LIN {X 0,Y 216.185,Z 698.743,A -85,B 0,C 180,E1 -24874.885,E2 -24874.885} C_VEL
LIN {X 0,Y 219.913,Z 693.734,A -85,B 0,C 180,E1 -24875.576,E2 -24875.576} C_VEL
LIN {X 0,Y 220.4,Z 693.095,A -85,B 0,C 180,E1 -24876,E2 -24876} C_VEL
LIN {X 0,Y 211.801,Z 704.873,A -85,B 0,C 180,E1 -24877.217,E2 -24877.217} C_VEL
LIN {X 0,Y 203.44,Z 714.464,A -85,B 0,C 180,E1 -24878.579,E2 -24878.579} C_VEL
LIN {X 0,Y 193.904,Z 723.929,A -85,B 0,C 180,E1 -24880.437,E2 -24880.437} C_VEL
LIN {X 0,Y 186.045,Z 730.716,A -85,B 0,C 180,E1 -24882.258,E2 -24882.258} C_VEL
LIN {X 0,Y 181.802,Z 733.879,A -85,B 0,C 180,E1 -24883.099,E2 -24883.099} C_VEL
LIN {X 0,Y 173.786,Z 738.72,A -85,B 0,C 180,E1 -24884.172,E2 -24884.172} C_VEL
LIN {X 0,Y 165.731,Z 742.885,A -85,B 0,C 180,E1 -24885.466,E2 -24885.466} C_VEL
LIN {X 0,Y 161.496,Z 744.973,A -85,B 0,C 180,E1 -24886.677,E2 -24886.677} C_VEL
LIN {X 0,Y 153.404,Z 748.777,A -85,B 0,C 180,E1 -24890.106,E2 -24890.106} C_VEL
LIN {X 0,Y 145.354,Z 751.765,A -85,B 0,C 180,E1 -24894.536,E2 -24894.536} C_VEL
LIN {X 0,Y 138.647,Z 753.472,A -85,B 0,C 180,E1 -24899.543,E2 -24899.543} C_VEL
LIN {X 0,Y 136.343,Z 754.019,A -85,B 0,C 180,E1 -24901.763,E2 -24901.763} C_VEL
LIN {X 0,Y 133.354,Z 759.17,A -85,B 0,C 180,E1 -24905.064,E2 -24905.064} C_VEL
LIN {X 0,Y 130.484,Z 764.543,A -85,B 0,C 180,E1 -24909.507,E2 -24909.507} C_VEL
LIN {X 0,Y 128.362,Z 768.722,A -85,B 0,C 180,E1 -24914.112,E2 -24914.112} C_VEL
LIN {X 0,Y 127.442,Z 770.931,A -85,B 0,C 180,E1 -24917.257,E2 -24917.257} C_VEL
LIN {X 0,Y 126.795,Z 772.646,A -85,B 0,C 180,E1 -24920.428,E2 -24920.428} C_VEL
LIN {X 0,Y 126.463,Z 773.951,A -85,B 0,C 180,E1 -24923.619,E2 -24923.619} C_VEL
LIN {X 0,Y 126.377,Z 774.859,A -85,B 0,C 180,E1 -24926.812,E2 -24926.812} C_VEL
LIN {X 0,Y 126.445,Z 775.338,A -85,B 0,C 180,E1 -24930,E2 -24930} C_VEL
LIN {X 0,Y 126.378,Z 775.387,A -85,B 0,C 180,E1 -24933.188,E2 -24933.188} C_VEL
LIN {X 0,Y 126.465,Z 775.046,A -85,B 0,C 180,E1 -24936.381,E2 -24936.381} C_VEL
LIN {X 0,Y 126.805,Z 774.317,A -85,B 0,C 180,E1 -24939.571,E2 -24939.571} C_VEL
LIN {X 0,Y 127.483,Z 773.149,A -85,B 0,C 180,E1 -24942.739,E2 -24942.739} C_VEL
LIN {X 0,Y 129.054,Z 770.628,A -85,B 0,C 180,E1 -24947.428,E2 -24947.428} C_VEL
LIN {X 0,Y 131.519,Z 767.102,A -85,B 0,C 180,E1 -24951.966,E2 -24951.966} C_VEL
LIN {X 0,Y 134.759,Z 762.463,A -85,B 0,C 180,E1 -24956.314,E2 -24956.314} C_VEL
LIN {X 0,Y 138.793,Z 756.345,A -85,B 0,C 180,E1 -24960.591,E2 -24960.591} C_VEL
LIN {X 0,Y 143.225,Z 749.227,A -85,B 0,C 180,E1 -24964.353,E2 -24964.353} C_VEL
LIN {X 0,Y 147.605,Z 741.745,A -85,B 0,C 180,E1 -24967.377,E2 -24967.377} C_VEL
LIN {X 0,Y 152.406,Z 732.671,A -85,B 0,C 180,E1 -24970.209,E2 -24970.209} C_VEL
LIN {X 0,Y 157.021,Z 722.567,A -85,B 0,C 180,E1 -24972.606,E2 -24972.606} C_VEL
LIN {X 0,Y 161.351,Z 711.381,A -85,B 0,C 180,E1 -24974.615,E2 -24974.615} C_VEL
LIN {X 0,Y 165.065,Z 699.776,A -85,B 0,C 180,E1 -24976.148,E2 -24976.148} C_VEL
LIN {X 0,Y 168.129,Z 687.035,A -85,B 0,C 180,E1 -24977.343,E2 -24977.343} C_VEL
LIN {X 0,Y 170.319,Z 673.92,A -85,B 0,C 180,E1 -24978.153,E2 -24978.153} C_VEL
LIN {X 0,Y 172.952,Z 640.488,A -85,B 0,C 180,E1 -24979.372,E2 -24979.372} C_VEL
LIN {X 0,Y 173.989,Z 625.56,A -85,B 0,C 180,E1 -24979.908,E2 -24979.908} C_VEL
LIN {X 0,Y 173.309,Z 610.583,A -85,B 0,C 180,E1 -24981.161,E2 -24981.161} C_VEL
LIN {X 0,Y 171.961,Z 606.297,A -85,B 0,C 180,E1 -24982.029,E2 -24982.029} C_VEL
LIN {X 0,Y 166.087,Z 595.425,A -85,B 0,C 180,E1 -24985.624,E2 -24985.624} C_VEL
LIN {X 0,Y 161.9,Z 588.541,A -85,B 0,C 180,E1 -24988.516,E2 -24988.516} C_VEL
LIN {X 0,Y 156.922,Z 580.807,A -85,B 0,C 180,E1 -24992.509,E2 -24992.509} C_VEL
LIN {X 0,Y 151.973,Z 573.867,A -85,B 0,C 180,E1 -24997.369,E2 -24997.369} C_VEL
LIN {X 0,Y 148.39,Z 569.165,A -85,B 0,C 180,E1 -25001.892,E2 -25001.892} C_VEL
LIN {X 0,Y 144.882,Z 564.63,A -85,B 0,C 180,E1 -25008.281,E2 -25008.281} C_VEL
LIN {X 0,Y 143.343,Z 562.894,A -85,B 0,C 180,E1 -25012.96,E2 -25012.96} C_VEL
LIN {X 0,Y 142.706,Z 561.543,A -85,B 0,C 180,E1 -25020.001,E2 -25020.001} C_VEL
LIN {X 0,Y 144.424,Z 564.073,A -85,B 0,C 180,E1 -25028.748,E2 -25028.748} C_VEL
LIN {X 0,Y 145.651,Z 565.845,A -85,B 0,C 180,E1 -25031.658,E2 -25031.658} C_VEL
LIN {X 0,Y 148.591,Z 569.435,A -85,B 0,C 180,E1 -25036.578,E2 -25036.578} C_VEL
LIN {X 0,Y 151.999,Z 574.091,A -85,B 0,C 180,E1 -25040.866,E2 -25040.866} C_VEL
LIN {X 0,Y 156.04,Z 579.845,A -85,B 0,C 180,E1 -25044.92,E2 -25044.92} C_VEL
LIN {X 0,Y 160.265,Z 586.52,A -85,B 0,C 180,E1 -25048.484,E2 -25048.484} C_VEL
LIN {X 0,Y 164.26,Z 593.492,A -85,B 0,C 180,E1 -25051.431,E2 -25051.431} C_VEL
LIN {X 0,Y 169.079,Z 602.683,A -85,B 0,C 180,E1 -25054.587,E2 -25054.587} C_VEL
LIN {X 0,Y 173.478,Z 612.626,A -85,B 0,C 180,E1 -25057.231,E2 -25057.231} C_VEL
LIN {X 0,Y 175.01,Z 616.566,A -85,B 0,C 180,E1 -25058.117,E2 -25058.117} C_VEL
LIN {X 0,Y 171.149,Z 666.622,A -85,B 0,C 180,E1 -25059.876,E2 -25059.876} C_VEL
LIN {X 0,Y 169.207,Z 679.283,A -85,B 0,C 180,E1 -25060.657,E2 -25060.657} C_VEL
LIN {X 0,Y 166.341,Z 692.094,A -85,B 0,C 180,E1 -25061.871,E2 -25061.871} C_VEL
LIN {X 0,Y 162.739,Z 704.293,A -85,B 0,C 180,E1 -25063.499,E2 -25063.499} C_VEL
LIN {X 0,Y 158.46,Z 716.072,A -85,B 0,C 180,E1 -25065.691,E2 -25065.691} C_VEL
LIN {X 0,Y 153.876,Z 726.187,A -85,B 0,C 180,E1 -25068.091,E2 -25068.091} C_VEL
LIN {X 0,Y 149.589,Z 734.459,A -85,B 0,C 180,E1 -25070.636,E2 -25070.636} C_VEL
LIN {X 0,Y 144.382,Z 743.398,A -85,B 0,C 180,E1 -25074.261,E2 -25074.261} C_VEL
LIN {X 0,Y 139.717,Z 750.589,A -85,B 0,C 180,E1 -25078.119,E2 -25078.119} C_VEL
LIN {X 0,Y 135.866,Z 756.334,A -85,B 0,C 180,E1 -25082.255,E2 -25082.255} C_VEL
LIN {X 0,Y 132.625,Z 760.828,A -85,B 0,C 180,E1 -25086.583,E2 -25086.583} C_VEL
LIN {X 0,Y 129.926,Z 764.224,A -85,B 0,C 180,E1 -25091.062,E2 -25091.062} C_VEL
LIN {X 0,Y 128.656,Z 765.907,A -85,B 0,C 180,E1 -25094.15,E2 -25094.15} C_VEL
LIN {X 0,Y 126.967,Z 768.068,A -85,B 0,C 180,E1 -25100.442,E2 -25100.442} C_VEL
LIN {X 0,Y 126.57,Z 768.541,A -85,B 0,C 180,E1 -25103.624,E2 -25103.624} C_VEL
LIN {X 0,Y 126.396,Z 768.598,A -85,B 0,C 180,E1 -25106.813,E2 -25106.813} C_VEL
LIN {X 0,Y 126.448,Z 768.276,A -85,B 0,C 180,E1 -25110,E2 -25110} C_VEL
LIN {X 0,Y 126.673,Z 767.577,A -85,B 0,C 180,E1 -25113.18,E2 -25113.18} C_VEL
LIN {X 0,Y 127.171,Z 766.448,A -85,B 0,C 180,E1 -25116.346,E2 -25116.346} C_VEL
LIN {X 0,Y 127.865,Z 764.905,A -85,B 0,C 180,E1 -25119.491,E2 -25119.491} C_VEL
LIN {X 0,Y 129.44,Z 761.796,A -85,B 0,C 180,E1 -25124.142,E2 -25124.142} C_VEL
LIN {X 0,Y 131.76,Z 757.626,A -85,B 0,C 180,E1 -25128.665,E2 -25128.665} C_VEL
LIN {X 0,Y 135.359,Z 751.288,A -85,B 0,C 180,E1 -25133.727,E2 -25133.727} C_VEL
LIN {X 0,Y 139.234,Z 744.3,A -85,B 0,C 180,E1 -25137.833,E2 -25137.833} C_VEL
LIN {X 0,Y 142.846,Z 737.187,A -85,B 0,C 180,E1 -25141.104,E2 -25141.104} C_VEL
LIN {X 0,Y 146.926,Z 728.562,A -85,B 0,C 180,E1 -25144.196,E2 -25144.196} C_VEL
LIN {X 0,Y 151.424,Z 717.961,A -85,B 0,C 180,E1 -25147.11,E2 -25147.11} C_VEL
LIN {X 0,Y 155.207,Z 707.284,A -85,B 0,C 180,E1 -25149.34,E2 -25149.34} C_VEL
LIN {X 0,Y 158.387,Z 696.357,A -85,B 0,C 180,E1 -25151.088,E2 -25151.088} C_VEL
LIN {X 0,Y 161.049,Z 684.52,A -85,B 0,C 180,E1 -25152.519,E2 -25152.519} C_VEL
LIN {X 0,Y 163.163,Z 671.837,A -85,B 0,C 180,E1 -25153.564,E2 -25153.564} C_VEL
LIN {X 0,Y 163.485,Z 668.976,A -85,B 0,C 180,E1 -25153.748,E2 -25153.748} C_VEL
LIN {X 0,Y 158.483,Z 675.492,A -85,B 0,C 180,E1 -25154.802,E2 -25154.802} C_VEL
LIN {X 0,Y 154.044,Z 679.517,A -85,B 0,C 180,E1 -25155.946,E2 -25155.946} C_VEL
LIN {X 0,Y 150.517,Z 681.416,A -85,B 0,C 180,E1 -25157.089,E2 -25157.089} C_VEL
LIN {X 0,Y 148.102,Z 682.143,A -85,B 0,C 180,E1 -25158.024,E2 -25158.024} C_VEL
LIN {X 0,Y 144.654,Z 685.261,A -85,B 0,C 180,E1 -25159.011,E2 -25159.011} C_VEL
LIN {X 0,Y 142.006,Z 686.87,A -85,B 0,C 180,E1 -25159.955,E2 -25159.955} C_VEL
LIN {X 0,Y 137.552,Z 687.512,A -85,B 0,C 180,E1 -25162.183,E2 -25162.183} C_VEL
LIN {X 0,Y 135.22,Z 689.383,A -85,B 0,C 180,E1 -25163.06,E2 -25163.06} C_VEL
LIN {X 0,Y 132.53,Z 690.745,A -85,B 0,C 180,E1 -25164.314,E2 -25164.314} C_VEL
LIN {X 0,Y 130.773,Z 690.191,A -85,B 0,C 180,E1 -25165.646,E2 -25165.646} C_VEL
LIN {X 0,Y 130.524,Z 688.78,A -85,B 0,C 180,E1 -25166.27,E2 -25166.27} C_VEL
LIN {X 0,Y 129.203,Z 698.323,A -85,B 0,C 180,E1 -25169.79,E2 -25169.79} C_VEL
LIN {X 0,Y 128.116,Z 707.573,A -85,B 0,C 180,E1 -25173.968,E2 -25173.968} C_VEL
LIN {X 0,Y 127.245,Z 716.39,A -85,B 0,C 180,E1 -25178.908,E2 -25178.908} C_VEL
LIN {X 0,Y 126.947,Z 723.62,A -85,B 0,C 180,E1 -25183.929,E2 -25183.929} C_VEL
LIN {X 0,Y 127.428,Z 729.309,A -85,B 0,C 180,E1 -25188.869,E2 -25188.869} C_VEL
LIN {X 0,Y 128.697,Z 733.847,A -85,B 0,C 180,E1 -25193.729,E2 -25193.729} C_VEL
LIN {X 0,Y 130.813,Z 737.363,A -85,B 0,C 180,E1 -25198.46,E2 -25198.46} C_VEL
LIN {X 0,Y 133.802,Z 739.916,A -85,B 0,C 180,E1 -25203.01,E2 -25203.01} C_VEL
LIN {X 0,Y 139.056,Z 742.012,A -85,B 0,C 180,E1 -25208.72,E2 -25208.72} C_VEL
LIN {X 0,Y 145.663,Z 742.543,A -85,B 0,C 180,E1 -25213.959,E2 -25213.959} C_VEL
LIN {X 0,Y 153.587,Z 741.587,A -85,B 0,C 180,E1 -25218.681,E2 -25218.681} C_VEL
LIN {X 0,Y 157.949,Z 740.525,A -85,B 0,C 180,E1 -25220.852,E2 -25220.852} C_VEL
LIN {X 0,Y 167.464,Z 737.157,A -85,B 0,C 180,E1 -25224.813,E2 -25224.813} C_VEL
LIN {X 0,Y 174.595,Z 733.792,A -85,B 0,C 180,E1 -25227.268,E2 -25227.268} C_VEL
LIN {X 0,Y 183.329,Z 728.781,A -85,B 0,C 180,E1 -25229.891,E2 -25229.891} C_VEL
LIN {X 0,Y 193.191,Z 721.838,A -85,B 0,C 180,E1 -25232.354,E2 -25232.354} C_VEL
LIN {X 0,Y 202.577,Z 713.844,A -85,B 0,C 180,E1 -25234.376,E2 -25234.376} C_VEL
LIN {X 0,Y 207.029,Z 709.49,A -85,B 0,C 180,E1 -25235.246,E2 -25235.246} C_VEL
LIN {X 0,Y 207.737,Z 708.837,A -85,B 0,C 180,E1 -25235.715,E2 -25235.715} C_VEL
LIN {X 0,Y 199.089,Z 717.814,A -85,B 0,C 180,E1 -25237.063,E2 -25237.063} C_VEL
LIN {X 0,Y 189.489,Z 726.349,A -85,B 0,C 180,E1 -25238.844,E2 -25238.844} C_VEL
LIN {X 0,Y 180.918,Z 732.987,A -85,B 0,C 180,E1 -25240.757,E2 -25240.757} C_VEL
LIN {X 0,Y 172.816,Z 738.494,A -85,B 0,C 180,E1 -25242.946,E2 -25242.946} C_VEL
LIN {X 0,Y 162.617,Z 744.408,A -85,B 0,C 180,E1 -25246.253,E2 -25246.253} C_VEL
LIN {X 0,Y 161.496,Z 744.973,A -85,B 0,C 180,E1 -25246.677,E2 -25246.677} C_VEL
LIN {X 0,Y 157.27,Z 746.892,A -85,B 0,C 180,E1 -25248.013,E2 -25248.013} C_VEL
LIN {X 0,Y 149.231,Z 749.489,A -85,B 0,C 180,E1 -25249.972,E2 -25249.972} C_VEL
LIN {X 0,Y 141.458,Z 751.288,A -85,B 0,C 180,E1 -25252.249,E2 -25252.249} C_VEL
LIN {X 0,Y 137.747,Z 752.026,A -85,B 0,C 180,E1 -25254.085,E2 -25254.085} C_VEL
LIN {X 0,Y 130.466,Z 753.197,A -85,B 0,C 180,E1 -25259.965,E2 -25259.965} C_VEL
LIN {X 0,Y 126.924,Z 758.914,A -85,B 0,C 180,E1 -25263.707,E2 -25263.707} C_VEL
LIN {X 0,Y 123.84,Z 764.299,A -85,B 0,C 180,E1 -25268.354,E2 -25268.354} C_VEL
LIN {X 0,Y 121.494,Z 768.49,A -85,B 0,C 180,E1 -25273.188,E2 -25273.188} C_VEL
LIN {X 0,Y 120.496,Z 770.707,A -85,B 0,C 180,E1 -25276.509,E2 -25276.509} C_VEL
LIN {X 0,Y 119.784,Z 772.431,A -85,B 0,C 180,E1 -25279.862,E2 -25279.862} C_VEL
LIN {X 0,Y 119.408,Z 773.742,A -85,B 0,C 180,E1 -25283.24,E2 -25283.24} C_VEL
LIN {X 0,Y 119.284,Z 774.655,A -85,B 0,C 180,E1 -25286.622,E2 -25286.622} C_VEL
LIN {X 0,Y 119.36,Z 775.144,A -85,B 0,C 180,E1 -25290,E2 -25290} C_VEL
LIN {X 0,Y 119.284,Z 775.198,A -85,B 0,C 180,E1 -25293.378,E2 -25293.378} C_VEL
LIN {X 0,Y 119.41,Z 774.862,A -85,B 0,C 180,E1 -25296.76,E2 -25296.76} C_VEL
LIN {X 0,Y 119.796,Z 774.139,A -85,B 0,C 180,E1 -25300.137,E2 -25300.137} C_VEL
LIN {X 0,Y 120.54,Z 772.982,A -85,B 0,C 180,E1 -25303.486,E2 -25303.486} C_VEL
LIN {X 0,Y 121.614,Z 771.4,A -85,B 0,C 180,E1 -25306.795,E2 -25306.795} C_VEL
LIN {X 0,Y 123.946,Z 768.227,A -85,B 0,C 180,E1 -25311.626,E2 -25311.626} C_VEL
LIN {X 0,Y 127.159,Z 763.988,A -85,B 0,C 180,E1 -25316.241,E2 -25316.241} C_VEL
LIN {X 0,Y 131.054,Z 758.726,A -85,B 0,C 180,E1 -25320.477,E2 -25320.477} C_VEL
LIN {X 0,Y 135.695,Z 751.765,A -85,B 0,C 180,E1 -25324.73,E2 -25324.73} C_VEL
LIN {X 0,Y 140.091,Z 744.835,A -85,B 0,C 180,E1 -25327.918,E2 -25327.918} C_VEL
LIN {X 0,Y 144.997,Z 736.473,A -85,B 0,C 180,E1 -25330.869,E2 -25330.869} C_VEL
LIN {X 0,Y 150.218,Z 726.13,A -85,B 0,C 180,E1 -25333.635,E2 -25333.635} C_VEL
LIN {X 0,Y 154.646,Z 715.905,A -85,B 0,C 180,E1 -25335.705,E2 -25335.705} C_VEL
LIN {X 0,Y 158.747,Z 704.702,A -85,B 0,C 180,E1 -25337.392,E2 -25337.392} C_VEL
LIN {X 0,Y 162.051,Z 693.189,A -85,B 0,C 180,E1 -25338.66,E2 -25338.66} C_VEL
LIN {X 0,Y 164.827,Z 680.09,A -85,B 0,C 180,E1 -25339.654,E2 -25339.654} C_VEL
LIN {X 0,Y 166.451,Z 667.33,A -85,B 0,C 180,E1 -25340.29,E2 -25340.29} C_VEL
LIN {X 0,Y 169.548,Z 626.44,A -85,B 0,C 180,E1 -25341.725,E2 -25341.725} C_VEL
LIN {X 0,Y 169.045,Z 613.188,A -85,B 0,C 180,E1 -25342.87,E2 -25342.87} C_VEL
LIN {X 0,Y 168.021,Z 610.42,A -85,B 0,C 180,E1 -25343.547,E2 -25343.547} C_VEL
LIN {X 0,Y 162.766,Z 600.331,A -85,B 0,C 180,E1 -25347.032,E2 -25347.032} C_VEL
LIN {X 0,Y 158.935,Z 593.804,A -85,B 0,C 180,E1 -25349.894,E2 -25349.894} C_VEL
LIN {X 0,Y 154.557,Z 586.727,A -85,B 0,C 180,E1 -25353.683,E2 -25353.683} C_VEL
LIN {X 0,Y 149.975,Z 580.077,A -85,B 0,C 180,E1 -25358.525,E2 -25358.525} C_VEL
LIN {X 0,Y 146.968,Z 575.882,A -85,B 0,C 180,E1 -25362.61,E2 -25362.61} C_VEL
LIN {X 0,Y 143.672,Z 571.382,A -85,B 0,C 180,E1 -25369.074,E2 -25369.074} C_VEL
LIN {X 0,Y 142.186,Z 569.639,A -85,B 0,C 180,E1 -25374.327,E2 -25374.327} C_VEL
LIN {X 0,Y 141.838,Z 568.612,A -85,B 0,C 180,E1 -25380.001,E2 -25380.001} C_VEL
LIN {X 0,Y 143.429,Z 571.071,A -85,B 0,C 180,E1 -25388.454,E2 -25388.454} C_VEL
LIN {X 0,Y 146.966,Z 575.845,A -85,B 0,C 180,E1 -25395.561,E2 -25395.561} C_VEL
LIN {X 0,Y 150.18,Z 580.528,A -85,B 0,C 180,E1 -25399.923,E2 -25399.923} C_VEL
LIN {X 0,Y 153.823,Z 585.93,A -85,B 0,C 180,E1 -25403.833,E2 -25403.833} C_VEL
LIN {X 0,Y 157.544,Z 592.09,A -85,B 0,C 180,E1 -25407.211,E2 -25407.211} C_VEL
LIN {X 0,Y 161.268,Z 598.852,A -85,B 0,C 180,E1 -25410.168,E2 -25410.168} C_VEL
LIN {X 0,Y 165.372,Z 607.004,A -85,B 0,C 180,E1 -25413.076,E2 -25413.076} C_VEL
LIN {X 0,Y 169.182,Z 615.779,A -85,B 0,C 180,E1 -25415.562,E2 -25415.562} C_VEL
LIN {X 0,Y 170.475,Z 619.097,A -85,B 0,C 180,E1 -25416.372,E2 -25416.372} C_VEL
LIN {X 0,Y 166.57,Z 667.069,A -85,B 0,C 180,E1 -25418.052,E2 -25418.052} C_VEL
LIN {X 0,Y 164.45,Z 680.046,A -85,B 0,C 180,E1 -25418.861,E2 -25418.861} C_VEL
LIN {X 0,Y 161.396,Z 693.035,A -85,B 0,C 180,E1 -25420.116,E2 -25420.116} C_VEL
LIN {X 0,Y 157.866,Z 704.424,A -85,B 0,C 180,E1 -25421.657,E2 -25421.657} C_VEL
LIN {X 0,Y 153.449,Z 716.071,A -85,B 0,C 180,E1 -25423.835,E2 -25423.835} C_VEL
LIN {X 0,Y 148.67,Z 726.22,A -85,B 0,C 180,E1 -25426.264,E2 -25426.264} C_VEL
LIN {X 0,Y 144.158,Z 734.522,A -85,B 0,C 180,E1 -25428.842,E2 -25428.842} C_VEL
LIN {X 0,Y 138.67,Z 743.491,A -85,B 0,C 180,E1 -25432.543,E2 -25432.543} C_VEL
LIN {X 0,Y 133.696,Z 750.699,A -85,B 0,C 180,E1 -25436.5,E2 -25436.5} C_VEL
LIN {X 0,Y 129.599,Z 756.46,A -85,B 0,C 180,E1 -25440.788,E2 -25440.788} C_VEL
LIN {X 0,Y 126.113,Z 760.971,A -85,B 0,C 180,E1 -25445.295,E2 -25445.295} C_VEL
LIN {X 0,Y 123.202,Z 764.38,A -85,B 0,C 180,E1 -25449.986,E2 -25449.986} C_VEL
LIN {X 0,Y 121.813,Z 766.073,A -85,B 0,C 180,E1 -25453.234,E2 -25453.234} C_VEL
LIN {X 0,Y 119.963,Z 768.245,A -85,B 0,C 180,E1 -25459.878,E2 -25459.878} C_VEL
LIN {X 0,Y 119.497,Z 768.73,A -85,B 0,C 180,E1 -25463.245,E2 -25463.245} C_VEL
LIN {X 0,Y 119.3,Z 768.792,A -85,B 0,C 180,E1 -25466.623,E2 -25466.623} C_VEL
LIN {X 0,Y 119.364,Z 768.475,A -85,B 0,C 180,E1 -25470,E2 -25470} C_VEL
LIN {X 0,Y 119.603,Z 767.782,A -85,B 0,C 180,E1 -25473.369,E2 -25473.369} C_VEL
LIN {X 0,Y 120.118,Z 766.665,A -85,B 0,C 180,E1 -25476.72,E2 -25476.72} C_VEL
LIN {X 0,Y 120.874,Z 765.127,A -85,B 0,C 180,E1 -25480.045,E2 -25480.045} C_VEL
LIN {X 0,Y 122.569,Z 762.03,A -85,B 0,C 180,E1 -25484.953,E2 -25484.953} C_VEL
LIN {X 0,Y 125.063,Z 757.873,A -85,B 0,C 180,E1 -25489.704,E2 -25489.704} C_VEL
LIN {X 0,Y 128.904,Z 751.549,A -85,B 0,C 180,E1 -25494.994,E2 -25494.994} C_VEL
LIN {X 0,Y 133.014,Z 744.582,A -85,B 0,C 180,E1 -25499.257,E2 -25499.257} C_VEL
LIN {X 0,Y 136.826,Z 737.487,A -85,B 0,C 180,E1 -25502.637,E2 -25502.637} C_VEL
LIN {X 0,Y 141.131,Z 728.881,A -85,B 0,C 180,E1 -25505.811,E2 -25505.811} C_VEL
LIN {X 0,Y 145.836,Z 718.309,A -85,B 0,C 180,E1 -25508.79,E2 -25508.79} C_VEL
LIN {X 0,Y 149.795,Z 707.679,A -85,B 0,C 180,E1 -25511.059,E2 -25511.059} C_VEL
LIN {X 0,Y 153.004,Z 697.218,A -85,B 0,C 180,E1 -25512.772,E2 -25512.772} C_VEL
LIN {X 0,Y 155.619,Z 686.362,A -85,B 0,C 180,E1 -25514.137,E2 -25514.137} C_VEL
LIN {X 0,Y 155.333,Z 685.227,A -85,B 0,C 180,E1 -25514.458,E2 -25514.458} C_VEL
LIN {X 0,Y 150.994,Z 687.583,A -85,B 0,C 180,E1 -25515.718,E2 -25515.718} C_VEL
LIN {X 0,Y 148.354,Z 688.642,A -85,B 0,C 180,E1 -25516.613,E2 -25516.613} C_VEL
LIN {X 0,Y 145.343,Z 691.001,A -85,B 0,C 180,E1 -25517.392,E2 -25517.392} C_VEL
LIN {X 0,Y 142.573,Z 692.606,A -85,B 0,C 180,E1 -25518.28,E2 -25518.28} C_VEL
LIN {X 0,Y 130.29,Z 697.275,A -85,B 0,C 180,E1 -25523.603,E2 -25523.603} C_VEL
LIN {X 0,Y 128.484,Z 696.83,A -85,B 0,C 180,E1 -25524.945,E2 -25524.945} C_VEL
LIN {X 0,Y 126.066,Z 698.186,A -85,B 0,C 180,E1 -25526.117,E2 -25526.117} C_VEL
LIN {X 0,Y 122.393,Z 698.352,A -85,B 0,C 180,E1 -25528.881,E2 -25528.881} C_VEL
LIN {X 0,Y 122.198,Z 697.195,A -85,B 0,C 180,E1 -25529.619,E2 -25529.619} C_VEL
LIN {X 0,Y 121.035,Z 707.059,A -85,B 0,C 180,E1 -25534.182,E2 -25534.182} C_VEL
LIN {X 0,Y 120.249,Z 714.901,A -85,B 0,C 180,E1 -25538.665,E2 -25538.665} C_VEL
LIN {X 0,Y 119.924,Z 722.221,A -85,B 0,C 180,E1 -25543.836,E2 -25543.836} C_VEL
LIN {X 0,Y 120.568,Z 729.182,A -85,B 0,C 180,E1 -25549.928,E2 -25549.928} C_VEL
LIN {X 0,Y 122.038,Z 733.869,A -85,B 0,C 180,E1 -25555.044,E2 -25555.044} C_VEL
LIN {X 0,Y 124.39,Z 737.506,A -85,B 0,C 180,E1 -25559.999,E2 -25559.999} C_VEL
LIN {X 0,Y 128.925,Z 740.989,A -85,B 0,C 180,E1 -25566.258,E2 -25566.258} C_VEL
LIN {X 0,Y 135.013,Z 742.877,A -85,B 0,C 180,E1 -25572.017,E2 -25572.017} C_VEL
LIN {X 0,Y 142.455,Z 743.295,A -85,B 0,C 180,E1 -25577.217,E2 -25577.217} C_VEL
LIN {X 0,Y 151.179,Z 742.222,A -85,B 0,C 180,E1 -25581.832,E2 -25581.832} C_VEL
LIN {X 0,Y 160.976,Z 739.526,A -85,B 0,C 180,E1 -25585.886,E2 -25585.886} C_VEL
LIN {X 0,Y 167.257,Z 737.184,A -85,B 0,C 180,E1 -25588.069,E2 -25588.069} C_VEL
LIN {X 0,Y 177.24,Z 732.347,A -85,B 0,C 180,E1 -25591.029,E2 -25591.029} C_VEL
LIN {X 0,Y 187.23,Z 726.357,A -85,B 0,C 180,E1 -25593.489,E2 -25593.489} C_VEL
LIN {X 0,Y 195.231,Z 720.529,A -85,B 0,C 180,E1 -25595.168,E2 -25595.168} C_VEL
LIN {X 0,Y 193.515,Z 722.027,A -85,B 0,C 180,E1 -25595.686,E2 -25595.686} C_VEL
LIN {X 0,Y 183.742,Z 729.75,A -85,B 0,C 180,E1 -25597.472,E2 -25597.472} C_VEL
LIN {X 0,Y 173.625,Z 736.504,A -85,B 0,C 180,E1 -25599.73,E2 -25599.73} C_VEL
LIN {X 0,Y 162.734,Z 742.633,A -85,B 0,C 180,E1 -25602.764,E2 -25602.764} C_VEL
LIN {X 0,Y 152.689,Z 747.236,A -85,B 0,C 180,E1 -25606.338,E2 -25606.338} C_VEL
LIN {X 0,Y 143.687,Z 750.487,A -85,B 0,C 180,E1 -25610.518,E2 -25610.518} C_VEL
LIN {X 0,Y 137.747,Z 752.026,A -85,B 0,C 180,E1 -25614.085,E2 -25614.085} C_VEL
LIN {X 0,Y 135.108,Z 752.43,A -85,B 0,C 180,E1 -25615.382,E2 -25615.382} C_VEL
LIN {X 0,Y 129.57,Z 752.929,A -85,B 0,C 180,E1 -25617.148,E2 -25617.148} C_VEL
LIN {X 0,Y 125.297,Z 753.941,A -85,B 0,C 180,E1 -25618.571,E2 -25618.571} C_VEL
LIN {X 0,Y 122.85,Z 755.393,A -85,B 0,C 180,E1 -25619.843,E2 -25619.843} C_VEL
LIN {X 0,Y 122.312,Z 756.05,A -85,B 0,C 180,E1 -25620.316,E2 -25620.316} C_VEL
LIN {X 0,Y 118.297,Z 762.42,A -85,B 0,C 180,E1 -25625.427,E2 -25625.427} C_VEL
LIN {X 0,Y 115.405,Z 767.004,A -85,B 0,C 180,E1 -25630.432,E2 -25630.432} C_VEL
LIN {X 0,Y 113.563,Z 770.482,A -85,B 0,C 180,E1 -25635.668,E2 -25635.668} C_VEL
LIN {X 0,Y 112.773,Z 772.216,A -85,B 0,C 180,E1 -25639.225,E2 -25639.225} C_VEL
LIN {X 0,Y 112.331,Z 773.532,A -85,B 0,C 180,E1 -25642.812,E2 -25642.812} C_VEL
LIN {X 0,Y 112.181,Z 774.45,A -85,B 0,C 180,E1 -25646.408,E2 -25646.408} C_VEL
LIN {X 0,Y 112.262,Z 774.951,A -85,B 0,C 180,E1 -25650,E2 -25650} C_VEL
LIN {X 0,Y 112.201,Z 775.01,A -85,B 0,C 180,E1 -25653.591,E2 -25653.591} C_VEL
LIN {X 0,Y 112.334,Z 774.679,A -85,B 0,C 180,E1 -25657.188,E2 -25657.188} C_VEL
LIN {X 0,Y 112.787,Z 773.961,A -85,B 0,C 180,E1 -25660.774,E2 -25660.774} C_VEL
LIN {X 0,Y 113.628,Z 772.814,A -85,B 0,C 180,E1 -25664.324,E2 -25664.324} C_VEL
LIN {X 0,Y 116.35,Z 769.251,A -85,B 0,C 180,E1 -25671.249,E2 -25671.249} C_VEL
LIN {X 0,Y 119.605,Z 765.396,A -85,B 0,C 180,E1 -25676.148,E2 -25676.148} C_VEL
LIN {X 0,Y 123.609,Z 760.4,A -85,B 0,C 180,E1 -25680.777,E2 -25680.777} C_VEL
LIN {X 0,Y 128.193,Z 754.1,A -85,B 0,C 180,E1 -25685.144,E2 -25685.144} C_VEL
LIN {X 0,Y 133.587,Z 746.216,A -85,B 0,C 180,E1 -25689.146,E2 -25689.146} C_VEL
LIN {X 0,Y 138.629,Z 738.181,A -85,B 0,C 180,E1 -25692.199,E2 -25692.199} C_VEL
LIN {X 0,Y 144.075,Z 728.378,A -85,B 0,C 180,E1 -25695.015,E2 -25695.015} C_VEL
LIN {X 0,Y 148.641,Z 718.711,A -85,B 0,C 180,E1 -25697.126,E2 -25697.126} C_VEL
LIN {X 0,Y 152.83,Z 708.224,A -85,B 0,C 180,E1 -25698.851,E2 -25698.851} C_VEL
LIN {X 0,Y 156.832,Z 695.661,A -85,B 0,C 180,E1 -25700.371,E2 -25700.371} C_VEL
LIN {X 0,Y 159.832,Z 683.032,A -85,B 0,C 180,E1 -25701.43,E2 -25701.43} C_VEL
LIN {X 0,Y 161.868,Z 669.56,A -85,B 0,C 180,E1 -25702.144,E2 -25702.144} C_VEL
LIN {X 0,Y 165.27,Z 627.482,A -85,B 0,C 180,E1 -25703.633,E2 -25703.633} C_VEL
LIN {X 0,Y 164.927,Z 615.979,A -85,B 0,C 180,E1 -25704.658,E2 -25704.658} C_VEL
LIN {X 0,Y 160.06,Z 606.16,A -85,B 0,C 180,E1 -25708.111,E2 -25708.111} C_VEL
LIN {X 0,Y 156.374,Z 599.616,A -85,B 0,C 180,E1 -25711.058,E2 -25711.058} C_VEL
LIN {X 0,Y 152.321,Z 592.753,A -85,B 0,C 180,E1 -25714.828,E2 -25714.828} C_VEL
LIN {X 0,Y 148.379,Z 586.728,A -85,B 0,C 180,E1 -25719.283,E2 -25719.283} C_VEL
LIN {X 0,Y 145.57,Z 582.595,A -85,B 0,C 180,E1 -25723.343,E2 -25723.343} C_VEL
LIN {X 0,Y 142.552,Z 578.205,A -85,B 0,C 180,E1 -25729.706,E2 -25729.706} C_VEL
LIN {X 0,Y 141.112,Z 576.378,A -85,B 0,C 180,E1 -25735.716,E2 -25735.716} C_VEL
LIN {X 0,Y 140.973,Z 575.661,A -85,B 0,C 180,E1 -25740.001,E2 -25740.001} C_VEL
LIN {X 0,Y 142.468,Z 578.104,A -85,B 0,C 180,E1 -25748.243,E2 -25748.243} C_VEL
LIN {X 0,Y 145.584,Z 582.605,A -85,B 0,C 180,E1 -25754.861,E2 -25754.861} C_VEL
LIN {X 0,Y 148.43,Z 586.963,A -85,B 0,C 180,E1 -25758.986,E2 -25758.986} C_VEL
LIN {X 0,Y 151.765,Z 592.169,A -85,B 0,C 180,E1 -25762.821,E2 -25762.821} C_VEL
LIN {X 0,Y 155.923,Z 599.381,A -85,B 0,C 180,E1 -25766.792,E2 -25766.792} C_VEL
LIN {X 0,Y 160.194,Z 607.894,A -85,B 0,C 180,E1 -25770.301,E2 -25770.301} C_VEL
LIN {X 0,Y 164.041,Z 616.447,A -85,B 0,C 180,E1 -25773.112,E2 -25773.112} C_VEL
LIN {X 0,Y 166.048,Z 621.666,A -85,B 0,C 180,E1 -25774.508,E2 -25774.508} C_VEL
LIN {X 0,Y 162.212,Z 666.883,A -85,B 0,C 180,E1 -25776.086,E2 -25776.086} C_VEL
LIN {X 0,Y 160.115,Z 679.693,A -85,B 0,C 180,E1 -25776.876,E2 -25776.876} C_VEL
LIN {X 0,Y 156.912,Z 692.892,A -85,B 0,C 180,E1 -25778.132,E2 -25778.132} C_VEL
LIN {X 0,Y 153.13,Z 704.629,A -85,B 0,C 180,E1 -25779.707,E2 -25779.707} C_VEL
LIN {X 0,Y 148.606,Z 716.072,A -85,B 0,C 180,E1 -25781.854,E2 -25781.854} C_VEL
LIN {X 0,Y 143.628,Z 726.254,A -85,B 0,C 180,E1 -25784.306,E2 -25784.306} C_VEL
LIN {X 0,Y 138.876,Z 734.584,A -85,B 0,C 180,E1 -25786.908,E2 -25786.908} C_VEL
LIN {X 0,Y 133.074,Z 743.583,A -85,B 0,C 180,E1 -25790.674,E2 -25790.674} C_VEL
LIN {X 0,Y 127.813,Z 750.809,A -85,B 0,C 180,E1 -25794.736,E2 -25794.736} C_VEL
LIN {X 0,Y 123.429,Z 756.586,A -85,B 0,C 180,E1 -25799.173,E2 -25799.173} C_VEL
LIN {X 0,Y 119.673,Z 761.113,A -85,B 0,C 180,E1 -25803.868,E2 -25803.868} C_VEL
LIN {X 0,Y 116.527,Z 764.535,A -85,B 0,C 180,E1 -25808.785,E2 -25808.785} C_VEL
LIN {X 0,Y 115.012,Z 766.238,A -85,B 0,C 180,E1 -25812.21,E2 -25812.21} C_VEL
LIN {X 0,Y 113.838,Z 767.525,A -85,B 0,C 180,E1 -25815.703,E2 -25815.703} C_VEL
LIN {X 0,Y 112.958,Z 768.422,A -85,B 0,C 180,E1 -25819.243,E2 -25819.243} C_VEL
LIN {X 0,Y 112.451,Z 768.917,A -85,B 0,C 180,E1 -25822.82,E2 -25822.82} C_VEL
LIN {X 0,Y 112.216,Z 768.985,A -85,B 0,C 180,E1 -25826.409,E2 -25826.409} C_VEL
LIN {X 0,Y 112.265,Z 768.674,A -85,B 0,C 180,E1 -25830,E2 -25830} C_VEL
LIN {X 0,Y 112.528,Z 767.986,A -85,B 0,C 180,E1 -25833.581,E2 -25833.581} C_VEL
LIN {X 0,Y 113.083,Z 766.881,A -85,B 0,C 180,E1 -25837.14,E2 -25837.14} C_VEL
LIN {X 0,Y 113.888,Z 765.35,A -85,B 0,C 180,E1 -25840.668,E2 -25840.668} C_VEL
LIN {X 0,Y 115.74,Z 762.263,A -85,B 0,C 180,E1 -25845.857,E2 -25845.857} C_VEL
LIN {X 0,Y 118.417,Z 758.118,A -85,B 0,C 180,E1 -25850.86,E2 -25850.86} C_VEL
LIN {X 0,Y 122.522,Z 751.81,A -85,B 0,C 180,E1 -25856.394,E2 -25856.394} C_VEL
LIN {X 0,Y 126.881,Z 744.863,A -85,B 0,C 180,E1 -25860.82,E2 -25860.82} C_VEL
LIN {X 0,Y 130.914,Z 737.786,A -85,B 0,C 180,E1 -25864.31,E2 -25864.31} C_VEL
LIN {X 0,Y 135.456,Z 729.2,A -85,B 0,C 180,E1 -25867.562,E2 -25867.562} C_VEL
LIN {X 0,Y 140.38,Z 718.654,A -85,B 0,C 180,E1 -25870.603,E2 -25870.603} C_VEL
LIN {X 0,Y 144.528,Z 708.073,A -85,B 0,C 180,E1 -25872.904,E2 -25872.904} C_VEL
LIN {X 0,Y 147.898,Z 697.658,A -85,B 0,C 180,E1 -25874.63,E2 -25874.63} C_VEL
LIN {X 0,Y 148.358,Z 696.01,A -85,B 0,C 180,E1 -25874.867,E2 -25874.867} C_VEL
LIN {X 0,Y 148.266,Z 695.014,A -85,B 0,C 180,E1 -25875.161,E2 -25875.161} C_VEL
LIN {X 0,Y 145.94,Z 696.635,A -85,B 0,C 180,E1 -25875.71,E2 -25875.71} C_VEL
LIN {X 0,Y 143.051,Z 698.229,A -85,B 0,C 180,E1 -25876.542,E2 -25876.542} C_VEL
LIN {X 0,Y 132.627,Z 702.056,A -85,B 0,C 180,E1 -25880.513,E2 -25880.513} C_VEL
LIN {X 0,Y 127.791,Z 703.645,A -85,B 0,C 180,E1 -25882.773,E2 -25882.773} C_VEL
LIN {X 0,Y 123.469,Z 704.523,A -85,B 0,C 180,E1 -25885.303,E2 -25885.303} C_VEL
LIN {X 0,Y 119.715,Z 704.687,A -85,B 0,C 180,E1 -25888.104,E2 -25888.104} C_VEL
LIN {X 0,Y 115.619,Z 706.201,A -85,B 0,C 180,E1 -25890.902,E2 -25890.902} C_VEL
LIN {X 0,Y 114.3,Z 705.701,A -85,B 0,C 180,E1 -25892.537,E2 -25892.537} C_VEL
LIN {X 0,Y 114.161,Z 704.62,A -85,B 0,C 180,E1 -25893.491,E2 -25893.491} C_VEL
LIN {X 0,Y 113.239,Z 714.235,A -85,B 0,C 180,E1 -25899.118,E2 -25899.118} C_VEL
LIN {X 0,Y 112.964,Z 721.894,A -85,B 0,C 180,E1 -25904.667,E2 -25904.667} C_VEL
LIN {X 0,Y 113.401,Z 727.148,A -85,B 0,C 180,E1 -25909.284,E2 -25909.284} C_VEL
LIN {X 0,Y 114.767,Z 732.319,A -85,B 0,C 180,E1 -25914.729,E2 -25914.729} C_VEL
LIN {X 0,Y 117.056,Z 736.458,A -85,B 0,C 180,E1 -25919.999,E2 -25919.999} C_VEL
LIN {X 0,Y 119.811,Z 739.267,A -85,B 0,C 180,E1 -25924.307,E2 -25924.307} C_VEL
LIN {X 0,Y 124.528,Z 741.975,A -85,B 0,C 180,E1 -25929.747,E2 -25929.747} C_VEL
LIN {X 0,Y 131.469,Z 743.744,A -85,B 0,C 180,E1 -25935.502,E2 -25935.502} C_VEL
LIN {X 0,Y 139.805,Z 744.064,A -85,B 0,C 180,E1 -25940.602,E2 -25940.602} C_VEL
LIN {X 0,Y 149.324,Z 742.842,A -85,B 0,C 180,E1 -25945.061,E2 -25945.061} C_VEL
LIN {X 0,Y 159.838,Z 740.097,A -85,B 0,C 180,E1 -25948.925,E2 -25948.925} C_VEL
LIN {X 0,Y 171.188,Z 735.651,A -85,B 0,C 180,E1 -25952.256,E2 -25952.256} C_VEL
LIN {X 0,Y 181.203,Z 730.507,A -85,B 0,C 180,E1 -25954.666,E2 -25954.666} C_VEL
LIN {X 0,Y 182.034,Z 730.033,A -85,B 0,C 180,E1 -25954.852,E2 -25954.852} C_VEL
LIN {X 0,Y 181.114,Z 730.719,A -85,B 0,C 180,E1 -25955.426,E2 -25955.426} C_VEL
LIN {X 0,Y 172.13,Z 736.321,A -85,B 0,C 180,E1 -25957.235,E2 -25957.235} C_VEL
LIN {X 0,Y 160.777,Z 742.23,A -85,B 0,C 180,E1 -25960.097,E2 -25960.097} C_VEL
LIN {X 0,Y 152.735,Z 745.724,A -85,B 0,C 180,E1 -25962.59,E2 -25962.59} C_VEL
LIN {X 0,Y 142.827,Z 749.147,A -85,B 0,C 180,E1 -25966.459,E2 -25966.459} C_VEL
LIN {X 0,Y 134.057,Z 751.323,A -85,B 0,C 180,E1 -25971.017,E2 -25971.017} C_VEL
LIN {X 0,Y 126.146,Z 752.309,A -85,B 0,C 180,E1 -25976.688,E2 -25976.688} C_VEL
LIN {X 0,Y 124.662,Z 752.436,A -85,B 0,C 180,E1 -25978.029,E2 -25978.029} C_VEL
LIN {X 0,Y 122.312,Z 756.05,A -85,B 0,C 180,E1 -25980.316,E2 -25980.316} C_VEL
LIN {X 0,Y 119.781,Z 759.084,A -85,B 0,C 180,E1 -25982.408,E2 -25982.408} C_VEL
LIN {X 0,Y 114.232,Z 763.437,A -85,B 0,C 180,E1 -25985.836,E2 -25985.836} C_VEL
LIN {X 0,Y 109.099,Z 767.13,A -85,B 0,C 180,E1 -25989.767,E2 -25989.767} C_VEL
LIN {X 0,Y 107.314,Z 769.015,A -85,B 0,C 180,E1 -25992.564,E2 -25992.564} C_VEL
LIN {X 0,Y 105.789,Z 772.001,A -85,B 0,C 180,E1 -25998.504,E2 -25998.504} C_VEL
LIN {X 0,Y 105.273,Z 773.322,A -85,B 0,C 180,E1 -26002.327,E2 -26002.327} C_VEL
LIN {X 0,Y 105.097,Z 774.246,A -85,B 0,C 180,E1 -26006.166,E2 -26006.166} C_VEL
LIN {X 0,Y 105.174,Z 774.757,A -85,B 0,C 180,E1 -26010,E2 -26010} C_VEL
LIN {X 0,Y 105.11,Z 774.821,A -85,B 0,C 180,E1 -26013.834,E2 -26013.834} C_VEL
LIN {X 0,Y 105.806,Z 773.782,A -85,B 0,C 180,E1 -26021.494,E2 -26021.494} C_VEL
LIN {X 0,Y 106.733,Z 772.647,A -85,B 0,C 180,E1 -26025.271,E2 -26025.271} C_VEL
LIN {X 0,Y 109.749,Z 769.095,A -85,B 0,C 180,E1 -26032.595,E2 -26032.595} C_VEL
LIN {X 0,Y 113.241,Z 765.252,A -85,B 0,C 180,E1 -26037.74,E2 -26037.74} C_VEL
LIN {X 0,Y 117.54,Z 760.271,A -85,B 0,C 180,E1 -26042.556,E2 -26042.556} C_VEL
LIN {X 0,Y 122.432,Z 753.991,A -85,B 0,C 180,E1 -26047.065,E2 -26047.065} C_VEL
LIN {X 0,Y 128.138,Z 746.127,A -85,B 0,C 180,E1 -26051.159,E2 -26051.159} C_VEL
LIN {X 0,Y 134.552,Z 736.35,A -85,B 0,C 180,E1 -26054.839,E2 -26054.839} C_VEL
LIN {X 0,Y 140.279,Z 726.076,A -85,B 0,C 180,E1 -26057.643,E2 -26057.643} C_VEL
LIN {X 0,Y 145.735,Z 714.525,A -85,B 0,C 180,E1 -26059.955,E2 -26059.955} C_VEL
LIN {X 0,Y 150.154,Z 702.965,A -85,B 0,C 180,E1 -26061.625,E2 -26061.625} C_VEL
LIN {X 0,Y 154.024,Z 689.772,A -85,B 0,C 180,E1 -26062.986,E2 -26062.986} C_VEL
LIN {X 0,Y 156.657,Z 677.088,A -85,B 0,C 180,E1 -26063.852,E2 -26063.852} C_VEL
LIN {X 0,Y 158.379,Z 661.943,A -85,B 0,C 180,E1 -26064.505,E2 -26064.505} C_VEL
LIN {X 0,Y 161.179,Z 628.419,A -85,B 0,C 180,E1 -26065.653,E2 -26065.653} C_VEL
LIN {X 0,Y 160.983,Z 619.538,A -85,B 0,C 180,E1 -26066.47,E2 -26066.47} C_VEL
LIN {X 0,Y 156.534,Z 610.369,A -85,B 0,C 180,E1 -26069.942,E2 -26069.942} C_VEL
LIN {X 0,Y 153.544,Z 604.81,A -85,B 0,C 180,E1 -26072.572,E2 -26072.572} C_VEL
LIN {X 0,Y 150.148,Z 598.772,A -85,B 0,C 180,E1 -26076.007,E2 -26076.007} C_VEL
LIN {X 0,Y 146.812,Z 593.358,A -85,B 0,C 180,E1 -26080.058,E2 -26080.058} C_VEL
LIN {X 0,Y 144.097,Z 589.188,A -85,B 0,C 180,E1 -26084.259,E2 -26084.259} C_VEL
LIN {X 0,Y 141.451,Z 585.016,A -85,B 0,C 180,E1 -26090.347,E2 -26090.347} C_VEL
LIN {X 0,Y 140.085,Z 583.014,A -85,B 0,C 180,E1 -26097.844,E2 -26097.844} C_VEL
LIN {X 0,Y 140.106,Z 582.719,A -85,B 0,C 180,E1 -26100.001,E2 -26100.001} C_VEL
LIN {X 0,Y 141.508,Z 585.142,A -85,B 0,C 180,E1 -26108.03,E2 -26108.03} C_VEL
LIN {X 0,Y 144.11,Z 589.144,A -85,B 0,C 180,E1 -26113.934,E2 -26113.934} C_VEL
LIN {X 0,Y 146.735,Z 593.443,A -85,B 0,C 180,E1 -26118.05,E2 -26118.05} C_VEL
LIN {X 0,Y 149.824,Z 598.558,A -85,B 0,C 180,E1 -26121.86,E2 -26121.86} C_VEL
LIN {X 0,Y 153.554,Z 605.397,A -85,B 0,C 180,E1 -26125.683,E2 -26125.683} C_VEL
LIN {X 0,Y 157.906,Z 614.575,A -85,B 0,C 180,E1 -26129.497,E2 -26129.497} C_VEL
LIN {X 0,Y 161.682,Z 623.89,A -85,B 0,C 180,E1 -26132.448,E2 -26132.448} C_VEL
LIN {X 0,Y 161.804,Z 624.245,A -85,B 0,C 180,E1 -26132.542,E2 -26132.542} C_VEL
LIN {X 0,Y 158.007,Z 667.371,A -85,B 0,C 180,E1 -26134.059,E2 -26134.059} C_VEL
LIN {X 0,Y 155.746,Z 680.39,A -85,B 0,C 180,E1 -26134.864,E2 -26134.864} C_VEL
LIN {X 0,Y 152.622,Z 692.749,A -85,B 0,C 180,E1 -26136.03,E2 -26136.03} C_VEL
LIN {X 0,Y 148.499,Z 705.05,A -85,B 0,C 180,E1 -26137.672,E2 -26137.672} C_VEL
LIN {X 0,Y 143.942,Z 716.072,A -85,B 0,C 180,E1 -26139.738,E2 -26139.738} C_VEL
LIN {X 0,Y 138.758,Z 726.288,A -85,B 0,C 180,E1 -26142.207,E2 -26142.207} C_VEL
LIN {X 0,Y 133.771,Z 734.645,A -85,B 0,C 180,E1 -26144.827,E2 -26144.827} C_VEL
LIN {X 0,Y 128.614,Z 742.335,A -85,B 0,C 180,E1 -26147.981,E2 -26147.981} C_VEL
LIN {X 0,Y 122.933,Z 749.823,A -85,B 0,C 180,E1 -26152.08,E2 -26152.08} C_VEL
LIN {X 0,Y 118.414,Z 755.382,A -85,B 0,C 180,E1 -26156.195,E2 -26156.195} C_VEL
LIN {X 0,Y 114.558,Z 759.859,A -85,B 0,C 180,E1 -26160.608,E2 -26160.608} C_VEL
LIN {X 0,Y 110.968,Z 763.646,A -85,B 0,C 180,E1 -26165.691,E2 -26165.691} C_VEL
LIN {X 0,Y 108.239,Z 766.404,A -85,B 0,C 180,E1 -26171.056,E2 -26171.056} C_VEL
LIN {X 0,Y 106.94,Z 767.697,A -85,B 0,C 180,E1 -26174.76,E2 -26174.76} C_VEL
LIN {X 0,Y 105.982,Z 768.599,A -85,B 0,C 180,E1 -26178.525,E2 -26178.525} C_VEL
LIN {X 0,Y 105.39,Z 769.105,A -85,B 0,C 180,E1 -26182.336,E2 -26182.336} C_VEL
LIN {X 0,Y 105.126,Z 769.179,A -85,B 0,C 180,E1 -26186.167,E2 -26186.167} C_VEL
LIN {X 0,Y 105.178,Z 768.873,A -85,B 0,C 180,E1 -26190,E2 -26190} C_VEL
LIN {X 0,Y 105.462,Z 768.191,A -85,B 0,C 180,E1 -26193.821,E2 -26193.821} C_VEL
LIN {X 0,Y 106.046,Z 767.097,A -85,B 0,C 180,E1 -26197.617,E2 -26197.617} C_VEL
LIN {X 0,Y 106.94,Z 765.571,A -85,B 0,C 180,E1 -26201.371,E2 -26201.371} C_VEL
LIN {X 0,Y 108.932,Z 762.497,A -85,B 0,C 180,E1 -26206.877,E2 -26206.877} C_VEL
LIN {X 0,Y 111.831,Z 758.364,A -85,B 0,C 180,E1 -26212.152,E2 -26212.152} C_VEL
LIN {X 0,Y 116.224,Z 752.069,A -85,B 0,C 180,E1 -26217.945,E2 -26217.945} C_VEL
LIN {X 0,Y 120.853,Z 745.145,A -85,B 0,C 180,E1 -26222.541,E2 -26222.541} C_VEL
LIN {X 0,Y 125.128,Z 738.085,A -85,B 0,C 180,E1 -26226.138,E2 -26226.138} C_VEL
LIN {X 0,Y 129.921,Z 729.518,A -85,B 0,C 180,E1 -26229.464,E2 -26229.464} C_VEL
LIN {X 0,Y 135.078,Z 718.997,A -85,B 0,C 180,E1 -26232.56,E2 -26232.56} C_VEL
LIN {X 0,Y 139.424,Z 708.466,A -85,B 0,C 180,E1 -26234.885,E2 -26234.885} C_VEL
LIN {X 0,Y 140.642,Z 704.807,A -85,B 0,C 180,E1 -26235.605,E2 -26235.605} C_VEL
LIN {X 0,Y 126.443,Z 709.533,A -85,B 0,C 180,E1 -26241.09,E2 -26241.09} C_VEL
LIN {X 0,Y 120.58,Z 710.677,A -85,B 0,C 180,E1 -26244.348,E2 -26244.348} C_VEL
LIN {X 0,Y 116.653,Z 710.992,A -85,B 0,C 180,E1 -26247.164,E2 -26247.164} C_VEL
LIN {X 0,Y 112.484,Z 712.296,A -85,B 0,C 180,E1 -26250.01,E2 -26250.01} C_VEL
LIN {X 0,Y 109.487,Z 712.051,A -85,B 0,C 180,E1 -26253.298,E2 -26253.298} C_VEL
LIN {X 0,Y 106.542,Z 712.371,A -85,B 0,C 180,E1 -26256.684,E2 -26256.684} C_VEL
LIN {X 0,Y 106.365,Z 711.188,A -85,B 0,C 180,E1 -26258.077,E2 -26258.077} C_VEL
LIN {X 0,Y 105.979,Z 719.012,A -85,B 0,C 180,E1 -26263.629,E2 -26263.629} C_VEL
LIN {X 0,Y 106.534,Z 726.463,A -85,B 0,C 180,E1 -26270.173,E2 -26270.173} C_VEL
LIN {X 0,Y 108.138,Z 732.159,A -85,B 0,C 180,E1 -26276.273,E2 -26276.273} C_VEL
LIN {X 0,Y 110.759,Z 736.465,A -85,B 0,C 180,E1 -26281.817,E2 -26281.817} C_VEL
LIN {X 0,Y 114.357,Z 739.825,A -85,B 0,C 180,E1 -26287.06,E2 -26287.06} C_VEL
LIN {X 0,Y 120.675,Z 742.94,A -85,B 0,C 180,E1 -26293.47,E2 -26293.47} C_VEL
LIN {X 0,Y 128.486,Z 744.607,A -85,B 0,C 180,E1 -26299.158,E2 -26299.158} C_VEL
LIN {X 0,Y 137.718,Z 744.814,A -85,B 0,C 180,E1 -26304.095,E2 -26304.095} C_VEL
LIN {X 0,Y 142.704,Z 744.357,A -85,B 0,C 180,E1 -26306.31,E2 -26306.31} C_VEL
LIN {X 0,Y 153.534,Z 742.279,A -85,B 0,C 180,E1 -26310.233,E2 -26310.233} C_VEL
LIN {X 0,Y 162.207,Z 739.692,A -85,B 0,C 180,E1 -26312.792,E2 -26312.792} C_VEL
LIN {X 0,Y 168.817,Z 737.201,A -85,B 0,C 180,E1 -26314.504,E2 -26314.504} C_VEL
LIN {X 0,Y 167.154,Z 738.164,A -85,B 0,C 180,E1 -26315.513,E2 -26315.513} C_VEL
LIN {X 0,Y 156.324,Z 743.12,A -85,B 0,C 180,E1 -26318.118,E2 -26318.118} C_VEL
LIN {X 0,Y 148.043,Z 746.21,A -85,B 0,C 180,E1 -26320.576,E2 -26320.576} C_VEL
LIN {X 0,Y 137.775,Z 749.182,A -85,B 0,C 180,E1 -26324.428,E2 -26324.428} C_VEL
LIN {X 0,Y 128.626,Z 750.923,A -85,B 0,C 180,E1 -26329.031,E2 -26329.031} C_VEL
LIN {X 0,Y 120.108,Z 751.482,A -85,B 0,C 180,E1 -26335.004,E2 -26335.004} C_VEL
LIN {X 0,Y 119.149,Z 751.536,A -85,B 0,C 180,E1 -26335.834,E2 -26335.834} C_VEL
LIN {X 0,Y 114.345,Z 758.403,A -85,B 0,C 180,E1 -26340.548,E2 -26340.548} C_VEL
LIN {X 0,Y 110.703,Z 763.812,A -85,B 0,C 180,E1 -26345.629,E2 -26345.629} C_VEL
LIN {X 0,Y 107.885,Z 768.024,A -85,B 0,C 180,E1 -26350.991,E2 -26350.991} C_VEL
LIN {X 0,Y 107.314,Z 769.015,A -85,B 0,C 180,E1 -26352.564,E2 -26352.564} C_VEL
LIN {X 0,Y 105.77,Z 770.698,A -85,B 0,C 180,E1 -26355.493,E2 -26355.493} C_VEL
LIN {X 0,Y 101.919,Z 772.738,A -85,B 0,C 180,E1 -26360.41,E2 -26360.41} C_VEL
LIN {X 0,Y 99.115,Z 773.817,A -85,B 0,C 180,E1 -26364.642,E2 -26364.642} C_VEL
LIN {X 0,Y 98.059,Z 774.349,A -85,B 0,C 180,E1 -26368.039,E2 -26368.039} C_VEL
LIN {X 0,Y 98.026,Z 774.461,A -85,B 0,C 180,E1 -26369.197,E2 -26369.197} C_VEL
LIN {X 0,Y 98.02,Z 774.633,A -85,B 0,C 180,E1 -26374.112,E2 -26374.112} C_VEL
LIN {X 0,Y 98.244,Z 774.312,A -85,B 0,C 180,E1 -26378.225,E2 -26378.225} C_VEL
LIN {X 0,Y 98.823,Z 773.604,A -85,B 0,C 180,E1 -26382.318,E2 -26382.318} C_VEL
LIN {X 0,Y 99.854,Z 772.479,A -85,B 0,C 180,E1 -26386.351,E2 -26386.351} C_VEL
LIN {X 0,Y 101.273,Z 770.914,A -85,B 0,C 180,E1 -26390.302,E2 -26390.302} C_VEL
LIN {X 0,Y 104.384,Z 767.778,A -85,B 0,C 180,E1 -26395.952,E2 -26395.952} C_VEL
LIN {X 0,Y 108.401,Z 763.577,A -85,B 0,C 180,E1 -26401.242,E2 -26401.242} C_VEL
LIN {X 0,Y 113.41,Z 757.944,A -85,B 0,C 180,E1 -26406.332,E2 -26406.332} C_VEL
LIN {X 0,Y 118.765,Z 751.445,A -85,B 0,C 180,E1 -26410.611,E2 -26410.611} C_VEL
LIN {X 0,Y 125.063,Z 743.038,A -85,B 0,C 180,E1 -26414.622,E2 -26414.622} C_VEL
LIN {X 0,Y 130.798,Z 734.385,A -85,B 0,C 180,E1 -26417.629,E2 -26417.629} C_VEL
LIN {X 0,Y 136.844,Z 723.74,A -85,B 0,C 180,E1 -26420.385,E2 -26420.385} C_VEL
LIN {X 0,Y 141.938,Z 713.057,A -85,B 0,C 180,E1 -26422.393,E2 -26422.393} C_VEL
LIN {X 0,Y 146.529,Z 701.118,A -85,B 0,C 180,E1 -26424.034,E2 -26424.034} C_VEL
LIN {X 0,Y 150.195,Z 688.685,A -85,B 0,C 180,E1 -26425.263,E2 -26425.263} C_VEL
LIN {X 0,Y 152.827,Z 676.091,A -85,B 0,C 180,E1 -26426.065,E2 -26426.065} C_VEL
LIN {X 0,Y 154.591,Z 660.419,A -85,B 0,C 180,E1 -26426.723,E2 -26426.723} C_VEL
LIN {X 0,Y 157.316,Z 628.666,A -85,B 0,C 180,E1 -26427.824,E2 -26427.824} C_VEL
LIN {X 0,Y 157.147,Z 623.001,A -85,B 0,C 180,E1 -26428.418,E2 -26428.418} C_VEL
LIN {X 0,Y 153.198,Z 614.556,A -85,B 0,C 180,E1 -26431.839,E2 -26431.839} C_VEL
LIN {X 0,Y 148.746,Z 605.932,A -85,B 0,C 180,E1 -26436.414,E2 -26436.414} C_VEL
LIN {X 0,Y 145.089,Z 599.747,A -85,B 0,C 180,E1 -26441.107,E2 -26441.107} C_VEL
LIN {X 0,Y 142.752,Z 595.919,A -85,B 0,C 180,E1 -26445.021,E2 -26445.021} C_VEL
LIN {X 0,Y 140.362,Z 591.879,A -85,B 0,C 180,E1 -26450.999,E2 -26450.999} C_VEL
LIN {X 0,Y 139.217,Z 590.076,A -85,B 0,C 180,E1 -26457.867,E2 -26457.867} C_VEL
LIN {X 0,Y 139.238,Z 589.788,A -85,B 0,C 180,E1 -26460.001,E2 -26460.001} C_VEL
LIN {X 0,Y 140.469,Z 592.04,A -85,B 0,C 180,E1 -26467.547,E2 -26467.547} C_VEL
LIN {X 0,Y 142.831,Z 596.022,A -85,B 0,C 180,E1 -26473.309,E2 -26473.309} C_VEL
LIN {X 0,Y 145.354,Z 600.427,A -85,B 0,C 180,E1 -26477.499,E2 -26477.499} C_VEL
LIN {X 0,Y 147.93,Z 604.915,A -85,B 0,C 180,E1 -26480.875,E2 -26480.875} C_VEL
LIN {X 0,Y 151.397,Z 611.747,A -85,B 0,C 180,E1 -26484.696,E2 -26484.696} C_VEL
LIN {X 0,Y 155.393,Z 620.815,A -85,B 0,C 180,E1 -26488.462,E2 -26488.462} C_VEL
LIN {X 0,Y 157.756,Z 626.911,A -85,B 0,C 180,E1 -26490.477,E2 -26490.477} C_VEL
LIN {X 0,Y 154.027,Z 667.62,A -85,B 0,C 180,E1 -26491.907,E2 -26491.907} C_VEL
LIN {X 0,Y 151.7,Z 680.578,A -85,B 0,C 180,E1 -26492.701,E2 -26492.701} C_VEL
LIN {X 0,Y 148.224,Z 693.693,A -85,B 0,C 180,E1 -26493.928,E2 -26493.928} C_VEL
LIN {X 0,Y 144.263,Z 705.006,A -85,B 0,C 180,E1 -26495.436,E2 -26495.436} C_VEL
LIN {X 0,Y 139.484,Z 716.098,A -85,B 0,C 180,E1 -26497.493,E2 -26497.493} C_VEL
LIN {X 0,Y 134.083,Z 726.323,A -85,B 0,C 180,E1 -26499.954,E2 -26499.954} C_VEL
LIN {X 0,Y 128.844,Z 734.707,A -85,B 0,C 180,E1 -26502.577,E2 -26502.577} C_VEL
LIN {X 0,Y 123.423,Z 742.422,A -85,B 0,C 180,E1 -26505.771,E2 -26505.771} C_VEL
LIN {X 0,Y 117.398,Z 749.933,A -85,B 0,C 180,E1 -26509.945,E2 -26509.945} C_VEL
LIN {X 0,Y 112.155,Z 755.932,A -85,B 0,C 180,E1 -26514.552,E2 -26514.552} C_VEL
LIN {X 0,Y 107.05,Z 761.396,A -85,B 0,C 180,E1 -26520.503,E2 -26520.503} C_VEL
LIN {X 0,Y 103.364,Z 764.844,A -85,B 0,C 180,E1 -26525.924,E2 -26525.924} C_VEL
LIN {X 0,Y 101.524,Z 766.57,A -85,B 0,C 180,E1 -26529.75,E2 -26529.75} C_VEL
LIN {X 0,Y 100.085,Z 767.868,A -85,B 0,C 180,E1 -26533.688,E2 -26533.688} C_VEL
LIN {X 0,Y 99.01,Z 768.777,A -85,B 0,C 180,E1 -26537.705,E2 -26537.705} C_VEL
LIN {X 0,Y 98.342,Z 769.292,A -85,B 0,C 180,E1 -26541.783,E2 -26541.783} C_VEL
LIN {X 0,Y 98.038,Z 769.373,A -85,B 0,C 180,E1 -26545.889,E2 -26545.889} C_VEL
LIN {X 0,Y 98.083,Z 769.073,A -85,B 0,C 180,E1 -26550,E2 -26550} C_VEL
LIN {X 0,Y 98.399,Z 768.395,A -85,B 0,C 180,E1 -26554.096,E2 -26554.096} C_VEL
LIN {X 0,Y 99.03,Z 767.313,A -85,B 0,C 180,E1 -26558.16,E2 -26558.16} C_VEL
LIN {X 0,Y 100,Z 765.792,A -85,B 0,C 180,E1 -26562.171,E2 -26562.171} C_VEL
LIN {X 0,Y 102.155,Z 762.731,A -85,B 0,C 180,E1 -26568.034,E2 -26568.034} C_VEL
LIN {X 0,Y 105.287,Z 758.61,A -85,B 0,C 180,E1 -26573.609,E2 -26573.609} C_VEL
LIN {X 0,Y 110.004,Z 752.328,A -85,B 0,C 180,E1 -26579.678,E2 -26579.678} C_VEL
LIN {X 0,Y 114.923,Z 745.427,A -85,B 0,C 180,E1 -26584.448,E2 -26584.448} C_VEL
LIN {X 0,Y 119.485,Z 738.384,A -85,B 0,C 180,E1 -26588.14,E2 -26588.14} C_VEL
LIN {X 0,Y 124.544,Z 729.837,A -85,B 0,C 180,E1 -26591.532,E2 -26591.532} C_VEL
LIN {X 0,Y 129.953,Z 719.34,A -85,B 0,C 180,E1 -26594.671,E2 -26594.671} C_VEL
LIN {X 0,Y 132.198,Z 714.407,A -85,B 0,C 180,E1 -26595.858,E2 -26595.858} C_VEL
LIN {X 0,Y 132.397,Z 712.983,A -85,B 0,C 180,E1 -26596.363,E2 -26596.363} C_VEL
LIN {X 0,Y 127.024,Z 714.63,A -85,B 0,C 180,E1 -26598.398,E2 -26598.398} C_VEL
LIN {X 0,Y 121.989,Z 715.874,A -85,B 0,C 180,E1 -26600.673,E2 -26600.673} C_VEL
LIN {X 0,Y 113.341,Z 717.033,A -85,B 0,C 180,E1 -26606.076,E2 -26606.076} C_VEL
LIN {X 0,Y 109.091,Z 718.195,A -85,B 0,C 180,E1 -26608.975,E2 -26608.975} C_VEL
LIN {X 0,Y 105.997,Z 717.97,A -85,B 0,C 180,E1 -26612.345,E2 -26612.345} C_VEL
LIN {X 0,Y 100.309,Z 718.582,A -85,B 0,C 180,E1 -26619.492,E2 -26619.492} C_VEL
LIN {X 0,Y 99.046,Z 717.395,A -85,B 0,C 180,E1 -26623.775,E2 -26623.775} C_VEL
LIN {X 0,Y 99.644,Z 725.39,A -85,B 0,C 180,E1 -26630.898,E2 -26630.898} C_VEL
LIN {X 0,Y 101.643,Z 731.908,A -85,B 0,C 180,E1 -26638.018,E2 -26638.018} C_VEL
LIN {X 0,Y 104.574,Z 736.361,A -85,B 0,C 180,E1 -26643.853,E2 -26643.853} C_VEL
LIN {X 0,Y 108.551,Z 739.897,A -85,B 0,C 180,E1 -26649.314,E2 -26649.314} C_VEL
LIN {X 0,Y 113.542,Z 742.555,A -85,B 0,C 180,E1 -26654.334,E2 -26654.334} C_VEL
LIN {X 0,Y 121.541,Z 744.848,A -85,B 0,C 180,E1 -26660.3,E2 -26660.3} C_VEL
LIN {X 0,Y 131.032,Z 745.706,A -85,B 0,C 180,E1 -26665.409,E2 -26665.409} C_VEL
LIN {X 0,Y 136.141,Z 745.575,A -85,B 0,C 180,E1 -26667.684,E2 -26667.684} C_VEL
LIN {X 0,Y 147.278,Z 744.199,A -85,B 0,C 180,E1 -26671.662,E2 -26671.662} C_VEL
LIN {X 0,Y 156.5,Z 742.065,A -85,B 0,C 180,E1 -26674.34,E2 -26674.34} C_VEL
LIN {X 0,Y 155.016,Z 742.769,A -85,B 0,C 180,E1 -26675.309,E2 -26675.309} C_VEL
LIN {X 0,Y 143.548,Z 746.583,A -85,B 0,C 180,E1 -26678.434,E2 -26678.434} C_VEL
LIN {X 0,Y 132.914,Z 749.096,A -85,B 0,C 180,E1 -26682.248,E2 -26682.248} C_VEL
LIN {X 0,Y 123.356,Z 750.418,A -85,B 0,C 180,E1 -26686.869,E2 -26686.869} C_VEL
LIN {X 0,Y 114.33,Z 750.527,A -85,B 0,C 180,E1 -26693.046,E2 -26693.046} C_VEL
LIN {X 0,Y 113.832,Z 750.611,A -85,B 0,C 180,E1 -26693.426,E2 -26693.426} C_VEL
LIN {X 0,Y 109.002,Z 757.144,A -85,B 0,C 180,E1 -26697.865,E2 -26697.865} C_VEL
LIN {X 0,Y 105.453,Z 761.918,A -85,B 0,C 180,E1 -26702.192,E2 -26702.192} C_VEL
LIN {X 0,Y 102.078,Z 766.531,A -85,B 0,C 180,E1 -26707.749,E2 -26707.749} C_VEL
LIN {X 0,Y 99.773,Z 770.03,A -85,B 0,C 180,E1 -26713.635,E2 -26713.635} C_VEL
LIN {X 0,Y 98.8,Z 771.785,A -85,B 0,C 180,E1 -26717.679,E2 -26717.679} C_VEL
LIN {X 0,Y 98.219,Z 773.112,A -85,B 0,C 180,E1 -26721.772,E2 -26721.772} C_VEL
LIN {X 0,Y 98.011,Z 774.041,A -85,B 0,C 180,E1 -26725.888,E2 -26725.888} C_VEL
LIN {X 0,Y 98.026,Z 774.461,A -85,B 0,C 180,E1 -26729.197,E2 -26729.197} C_VEL
LIN {X 0,Y 97.813,Z 774.676,A -85,B 0,C 180,E1 -26731.484,E2 -26731.484} C_VEL
LIN {X 0,Y 97.093,Z 774.745,A -85,B 0,C 180,E1 -26733.758,E2 -26733.758} C_VEL
LIN {X 0,Y 94.948,Z 774.464,A -85,B 0,C 180,E1 -26738.327,E2 -26738.327} C_VEL
LIN {X 0,Y 93.095,Z 773.616,A -85,B 0,C 180,E1 -26743.089,E2 -26743.089} C_VEL
LIN {X 0,Y 92.858,Z 772.6,A -85,B 0,C 180,E1 -26746.733,E2 -26746.733} C_VEL
LIN {X 0,Y 93.132,Z 772.188,A -85,B 0,C 180,E1 -26747.928,E2 -26747.928} C_VEL
LIN {X 0,Y 96.775,Z 768.785,A -85,B 0,C 180,E1 -26755.831,E2 -26755.831} C_VEL
LIN {X 0,Y 100.813,Z 764.965,A -85,B 0,C 180,E1 -26761.523,E2 -26761.523} C_VEL
LIN {X 0,Y 105.776,Z 760.01,A -85,B 0,C 180,E1 -26766.724,E2 -26766.724} C_VEL
LIN {X 0,Y 111.379,Z 753.77,A -85,B 0,C 180,E1 -26771.493,E2 -26771.493} C_VEL
LIN {X 0,Y 117.815,Z 745.949,A -85,B 0,C 180,E1 -26775.71,E2 -26775.71} C_VEL
LIN {X 0,Y 124.886,Z 736.22,A -85,B 0,C 180,E1 -26779.438,E2 -26779.438} C_VEL
LIN {X 0,Y 131.134,Z 726.023,A -85,B 0,C 180,E1 -26782.231,E2 -26782.231} C_VEL
LIN {X 0,Y 137.037,Z 714.545,A -85,B 0,C 180,E1 -26784.502,E2 -26784.502} C_VEL
LIN {X 0,Y 141.795,Z 703.145,A -85,B 0,C 180,E1 -26786.118,E2 -26786.118} C_VEL
LIN {X 0,Y 145.939,Z 690.128,A -85,B 0,C 180,E1 -26787.43,E2 -26787.43} C_VEL
LIN {X 0,Y 148.872,Z 677.228,A -85,B 0,C 180,E1 -26788.294,E2 -26788.294} C_VEL
LIN {X 0,Y 150.64,Z 663.524,A -85,B 0,C 180,E1 -26788.885,E2 -26788.885} C_VEL
LIN {X 0,Y 153.66,Z 629.562,A -85,B 0,C 180,E1 -26790.06,E2 -26790.06} C_VEL
LIN {X 0,Y 153.591,Z 626.842,A -85,B 0,C 180,E1 -26790.365,E2 -26790.365} C_VEL
LIN {X 0,Y 150.297,Z 619.371,A -85,B 0,C 180,E1 -26793.542,E2 -26793.542} C_VEL
LIN {X 0,Y 146.327,Z 611.389,A -85,B 0,C 180,E1 -26798.055,E2 -26798.055} C_VEL
LIN {X 0,Y 143.505,Z 606.274,A -85,B 0,C 180,E1 -26802.042,E2 -26802.042} C_VEL
LIN {X 0,Y 141.435,Z 602.623,A -85,B 0,C 180,E1 -26805.798,E2 -26805.798} C_VEL
LIN {X 0,Y 139.293,Z 598.73,A -85,B 0,C 180,E1 -26811.66,E2 -26811.66} C_VEL
LIN {X 0,Y 138.338,Z 596.981,A -85,B 0,C 180,E1 -26818.927,E2 -26818.927} C_VEL
LIN {X 0,Y 138.384,Z 597.055,A -85,B 0,C 180,E1 -26820.728,E2 -26820.728} C_VEL
LIN {X 0,Y 139.435,Z 598.984,A -85,B 0,C 180,E1 -26827.058,E2 -26827.058} C_VEL
LIN {X 0,Y 141.431,Z 602.601,A -85,B 0,C 180,E1 -26832.375,E2 -26832.375} C_VEL
LIN {X 0,Y 143.61,Z 606.674,A -85,B 0,C 180,E1 -26836.344,E2 -26836.344} C_VEL
LIN {X 0,Y 145.892,Z 610.898,A -85,B 0,C 180,E1 -26839.616,E2 -26839.616} C_VEL
LIN {X 0,Y 148.94,Z 617.294,A -85,B 0,C 180,E1 -26843.295,E2 -26843.295} C_VEL
LIN {X 0,Y 152.417,Z 625.74,A -85,B 0,C 180,E1 -26846.902,E2 -26846.902} C_VEL
LIN {X 0,Y 153.923,Z 629.775,A -85,B 0,C 180,E1 -26848.326,E2 -26848.326} C_VEL
LIN {X 0,Y 150.207,Z 668.406,A -85,B 0,C 180,E1 -26849.672,E2 -26849.672} C_VEL
LIN {X 0,Y 147.605,Z 681.892,A -85,B 0,C 180,E1 -26850.501,E2 -26850.501} C_VEL
LIN {X 0,Y 144.043,Z 694.629,A -85,B 0,C 180,E1 -26851.704,E2 -26851.704} C_VEL
LIN {X 0,Y 139.542,Z 706.657,A -85,B 0,C 180,E1 -26853.342,E2 -26853.342} C_VEL
LIN {X 0,Y 134.76,Z 717.117,A -85,B 0,C 180,E1 -26855.315,E2 -26855.315} C_VEL
LIN {X 0,Y 129.02,Z 727.398,A -85,B 0,C 180,E1 -26857.83,E2 -26857.83} C_VEL
LIN {X 0,Y 122.979,Z 736.429,A -85,B 0,C 180,E1 -26860.783,E2 -26860.783} C_VEL
LIN {X 0,Y 116.236,Z 745.192,A -85,B 0,C 180,E1 -26864.731,E2 -26864.731} C_VEL
LIN {X 0,Y 110.059,Z 752.232,A -85,B 0,C 180,E1 -26869.117,E2 -26869.117} C_VEL
LIN {X 0,Y 103.942,Z 758.607,A -85,B 0,C 180,E1 -26874.921,E2 -26874.921} C_VEL
LIN {X 0,Y 99.493,Z 762.789,A -85,B 0,C 180,E1 -26880.366,E2 -26880.366} C_VEL
LIN {X 0,Y 96.908,Z 764.997,A -85,B 0,C 180,E1 -26884.207,E2 -26884.207} C_VEL
LIN {X 0,Y 94.853,Z 766.737,A -85,B 0,C 180,E1 -26888.256,E2 -26888.256} C_VEL
LIN {X 0,Y 93.279,Z 768.04,A -85,B 0,C 180,E1 -26892.46,E2 -26892.46} C_VEL
LIN {X 0,Y 91.32,Z 769.477,A -85,B 0,C 180,E1 -26901.146,E2 -26901.146} C_VEL
LIN {X 0,Y 90.947,Z 769.568,A -85,B 0,C 180,E1 -26905.568,E2 -26905.568} C_VEL
LIN {X 0,Y 90.982,Z 769.272,A -85,B 0,C 180,E1 -26910,E2 -26910} C_VEL
LIN {X 0,Y 91.327,Z 768.6,A -85,B 0,C 180,E1 -26914.413,E2 -26914.413} C_VEL
LIN {X 0,Y 92.027,Z 767.528,A -85,B 0,C 180,E1 -26918.785,E2 -26918.785} C_VEL
LIN {X 0,Y 93.072,Z 766.014,A -85,B 0,C 180,E1 -26923.093,E2 -26923.093} C_VEL
LIN {X 0,Y 95.432,Z 762.964,A -85,B 0,C 180,E1 -26929.353,E2 -26929.353} C_VEL
LIN {X 0,Y 98.827,Z 758.856,A -85,B 0,C 180,E1 -26935.257,E2 -26935.257} C_VEL
LIN {X 0,Y 103.906,Z 752.586,A -85,B 0,C 180,E1 -26941.613,E2 -26941.613} C_VEL
LIN {X 0,Y 109.148,Z 745.709,A -85,B 0,C 180,E1 -26946.555,E2 -26946.555} C_VEL
LIN {X 0,Y 115.006,Z 737.09,A -85,B 0,C 180,E1 -26951.065,E2 -26951.065} C_VEL
LIN {X 0,Y 120.433,Z 728.25,A -85,B 0,C 180,E1 -26954.447,E2 -26954.447} C_VEL
LIN {X 0,Y 123.775,Z 722.106,A -85,B 0,C 180,E1 -26956.309,E2 -26956.309} C_VEL
LIN {X 0,Y 123.909,Z 720.494,A -85,B 0,C 180,E1 -26957.106,E2 -26957.106} C_VEL
LIN {X 0,Y 118.771,Z 721.632,A -85,B 0,C 180,E1 -26959.389,E2 -26959.389} C_VEL
LIN {X 0,Y 109.82,Z 722.821,A -85,B 0,C 180,E1 -26964.832,E2 -26964.832} C_VEL
LIN {X 0,Y 105.461,Z 723.873,A -85,B 0,C 180,E1 -26967.782,E2 -26967.782} C_VEL
LIN {X 0,Y 102.254,Z 723.674,A -85,B 0,C 180,E1 -26971.24,E2 -26971.24} C_VEL
LIN {X 0,Y 96.342,Z 724.265,A -85,B 0,C 180,E1 -26978.607,E2 -26978.607} C_VEL
LIN {X 0,Y 94.874,Z 723.418,A -85,B 0,C 180,E1 -26982.763,E2 -26982.763} C_VEL
LIN {X 0,Y 92.641,Z 724.283,A -85,B 0,C 180,E1 -26986.844,E2 -26986.844} C_VEL
LIN {X 0,Y 92.622,Z 723.152,A -85,B 0,C 180,E1 -26990.726,E2 -26990.726} C_VEL
LIN {X 0,Y 94.409,Z 729.764,A -85,B 0,C 180,E1 -26997.866,E2 -26997.866} C_VEL
LIN {X 0,Y 97.309,Z 734.759,A -85,B 0,C 180,E1 -27004.141,E2 -27004.141} C_VEL
LIN {X 0,Y 101.356,Z 738.746,A -85,B 0,C 180,E1 -27009.982,E2 -27009.982} C_VEL
LIN {X 0,Y 106.429,Z 741.884,A -85,B 0,C 180,E1 -27015.315,E2 -27015.315} C_VEL
LIN {X 0,Y 114.646,Z 744.794,A -85,B 0,C 180,E1 -27021.58,E2 -27021.58} C_VEL
LIN {X 0,Y 124.38,Z 746.306,A -85,B 0,C 180,E1 -27026.874,E2 -27026.874} C_VEL
LIN {X 0,Y 135.238,Z 746.342,A -85,B 0,C 180,E1 -27031.31,E2 -27031.31} C_VEL
LIN {X 0,Y 145.042,Z 745.285,A -85,B 0,C 180,E1 -27034.542,E2 -27034.542} C_VEL
LIN {X 0,Y 133.633,Z 747.958,A -85,B 0,C 180,E1 -27037.921,E2 -27037.921} C_VEL
LIN {X 0,Y 123.132,Z 749.446,A -85,B 0,C 180,E1 -27042.1,E2 -27042.1} C_VEL
LIN {X 0,Y 113.787,Z 749.802,A -85,B 0,C 180,E1 -27047.204,E2 -27047.204} C_VEL
LIN {X 0,Y 108.766,Z 749.641,A -85,B 0,C 180,E1 -27050.803,E2 -27050.803} C_VEL
LIN {X 0,Y 103.876,Z 755.789,A -85,B 0,C 180,E1 -27054.895,E2 -27054.895} C_VEL
LIN {X 0,Y 99.181,Z 761.667,A -85,B 0,C 180,E1 -27060.264,E2 -27060.264} C_VEL
LIN {X 0,Y 95.514,Z 766.293,A -85,B 0,C 180,E1 -27066.129,E2 -27066.129} C_VEL
LIN {X 0,Y 92.952,Z 769.804,A -85,B 0,C 180,E1 -27072.397,E2 -27072.397} C_VEL
LIN {X 0,Y 91.847,Z 771.569,A -85,B 0,C 180,E1 -27076.729,E2 -27076.729} C_VEL
LIN {X 0,Y 91.17,Z 772.901,A -85,B 0,C 180,E1 -27081.131,E2 -27081.131} C_VEL
LIN {X 0,Y 90.921,Z 773.837,A -85,B 0,C 180,E1 -27085.567,E2 -27085.567} C_VEL
LIN {X 0,Y 90.977,Z 774.367,A -85,B 0,C 180,E1 -27090,E2 -27090} C_VEL
LIN {X 0,Y 90.929,Z 774.444,A -85,B 0,C 180,E1 -27094.433,E2 -27094.433} C_VEL
LIN {X 0,Y 91.191,Z 774.128,A -85,B 0,C 180,E1 -27098.867,E2 -27098.867} C_VEL
LIN {X 0,Y 91.873,Z 773.425,A -85,B 0,C 180,E1 -27103.267,E2 -27103.267} C_VEL
LIN {X 0,Y 93.132,Z 772.188,A -85,B 0,C 180,E1 -27107.928,E2 -27107.928} C_VEL
LIN {X 0,Y 93.777,Z 770.955,A -85,B 0,C 180,E1 -27111.442,E2 -27111.442} C_VEL
LIN {X 0,Y 93.883,Z 768.431,A -85,B 0,C 180,E1 -27117.313,E2 -27117.313} C_VEL
LIN {X 0,Y 94.907,Z 765.276,A -85,B 0,C 180,E1 -27122.988,E2 -27122.988} C_VEL
LIN {X 0,Y 96.894,Z 762.96,A -85,B 0,C 180,E1 -27126.011,E2 -27126.011} C_VEL
LIN {X 0,Y 102.159,Z 757.809,A -85,B 0,C 180,E1 -27130.982,E2 -27130.982} C_VEL
LIN {X 0,Y 108.346,Z 751.232,A -85,B 0,C 180,E1 -27135.521,E2 -27135.521} C_VEL
LIN {X 0,Y 115.372,Z 742.881,A -85,B 0,C 180,E1 -27139.59,E2 -27139.59} C_VEL
LIN {X 0,Y 121.686,Z 734.276,A -85,B 0,C 180,E1 -27142.572,E2 -27142.572} C_VEL
LIN {X 0,Y 128.276,Z 723.688,A -85,B 0,C 180,E1 -27145.265,E2 -27145.265} C_VEL
LIN {X 0,Y 133.761,Z 713.122,A -85,B 0,C 180,E1 -27147.208,E2 -27147.208} C_VEL
LIN {X 0,Y 138.688,Z 701.3,A -85,B 0,C 180,E1 -27148.773,E2 -27148.773} C_VEL
LIN {X 0,Y 142.604,Z 689.054,A -85,B 0,C 180,E1 -27149.942,E2 -27149.942} C_VEL
LIN {X 0,Y 145.408,Z 676.865,A -85,B 0,C 180,E1 -27150.712,E2 -27150.712} C_VEL
LIN {X 0,Y 147.31,Z 662.318,A -85,B 0,C 180,E1 -27151.311,E2 -27151.311} C_VEL
LIN {X 0,Y 150.255,Z 630.642,A -85,B 0,C 180,E1 -27152.378,E2 -27152.378} C_VEL
LIN {X 0,Y 146.987,Z 623.121,A -85,B 0,C 180,E1 -27155.927,E2 -27155.927} C_VEL
LIN {X 0,Y 144.157,Z 617.033,A -85,B 0,C 180,E1 -27159.581,E2 -27159.581} C_VEL
LIN {X 0,Y 141.808,Z 612.546,A -85,B 0,C 180,E1 -27163.258,E2 -27163.258} C_VEL
LIN {X 0,Y 140.147,Z 609.313,A -85,B 0,C 180,E1 -27166.59,E2 -27166.59} C_VEL
LIN {X 0,Y 138.33,Z 605.739,A -85,B 0,C 180,E1 -27171.969,E2 -27171.969} C_VEL
LIN {X 0,Y 137.47,Z 604.042,A -85,B 0,C 180,E1 -27178.921,E2 -27178.921} C_VEL
LIN {X 0,Y 137.514,Z 604.137,A -85,B 0,C 180,E1 -27180.733,E2 -27180.733} C_VEL
LIN {X 0,Y 138.455,Z 606.036,A -85,B 0,C 180,E1 -27186.742,E2 -27186.742} C_VEL
LIN {X 0,Y 140.135,Z 609.31,A -85,B 0,C 180,E1 -27191.573,E2 -27191.573} C_VEL
LIN {X 0,Y 142.173,Z 613.44,A -85,B 0,C 180,E1 -27195.593,E2 -27195.593} C_VEL
LIN {X 0,Y 144.094,Z 617.321,A -85,B 0,C 180,E1 -27198.576,E2 -27198.576} C_VEL
LIN {X 0,Y 146.746,Z 623.318,A -85,B 0,C 180,E1 -27202.066,E2 -27202.066} C_VEL
LIN {X 0,Y 149.68,Z 630.971,A -85,B 0,C 180,E1 -27205.407,E2 -27205.407} C_VEL
LIN {X 0,Y 150.287,Z 632.67,A -85,B 0,C 180,E1 -27206.047,E2 -27206.047} C_VEL
LIN {X 0,Y 146.698,Z 668.68,A -85,B 0,C 180,E1 -27207.3,E2 -27207.3} C_VEL
LIN {X 0,Y 144.055,Z 681.949,A -85,B 0,C 180,E1 -27208.092,E2 -27208.092} C_VEL
LIN {X 0,Y 140.426,Z 694.498,A -85,B 0,C 180,E1 -27209.227,E2 -27209.227} C_VEL
LIN {X 0,Y 135.768,Z 706.615,A -85,B 0,C 180,E1 -27210.837,E2 -27210.837} C_VEL
LIN {X 0,Y 130.511,Z 717.621,A -85,B 0,C 180,E1 -27212.875,E2 -27212.875} C_VEL
LIN {X 0,Y 124.78,Z 727.438,A -85,B 0,C 180,E1 -27215.248,E2 -27215.248} C_VEL
LIN {X 0,Y 118.441,Z 736.502,A -85,B 0,C 180,E1 -27218.168,E2 -27218.168} C_VEL
LIN {X 0,Y 111.334,Z 745.286,A -85,B 0,C 180,E1 -27222.123,E2 -27222.123} C_VEL
LIN {X 0,Y 104.78,Z 752.347,A -85,B 0,C 180,E1 -27226.568,E2 -27226.568} C_VEL
LIN {X 0,Y 99.918,Z 757.095,A -85,B 0,C 180,E1 -27230.727,E2 -27230.727} C_VEL
LIN {X 0,Y 94.896,Z 761.678,A -85,B 0,C 180,E1 -27236.259,E2 -27236.259} C_VEL
LIN {X 0,Y 90.556,Z 765.151,A -85,B 0,C 180,E1 -27242.248,E2 -27242.248} C_VEL
LIN {X 0,Y 88.26,Z 766.903,A -85,B 0,C 180,E1 -27246.538,E2 -27246.538} C_VEL
LIN {X 0,Y 86.51,Z 768.212,A -85,B 0,C 180,E1 -27251.038,E2 -27251.038} C_VEL
LIN {X 0,Y 85.176,Z 769.131,A -85,B 0,C 180,E1 -27255.669,E2 -27255.669} C_VEL
LIN {X 0,Y 84.301,Z 769.663,A -85,B 0,C 180,E1 -27260.402,E2 -27260.402} C_VEL
LIN {X 0,Y 83.881,Z 769.761,A -85,B 0,C 180,E1 -27265.194,E2 -27265.194} C_VEL
LIN {X 0,Y 83.888,Z 769.471,A -85,B 0,C 180,E1 -27270,E2 -27270} C_VEL
LIN {X 0,Y 84.269,Z 768.804,A -85,B 0,C 180,E1 -27274.784,E2 -27274.784} C_VEL
LIN {X 0,Y 85.036,Z 767.743,A -85,B 0,C 180,E1 -27279.514,E2 -27279.514} C_VEL
LIN {X 0,Y 86.19,Z 766.236,A -85,B 0,C 180,E1 -27284.159,E2 -27284.159} C_VEL
LIN {X 0,Y 88.776,Z 763.197,A -85,B 0,C 180,E1 -27290.869,E2 -27290.869} C_VEL
LIN {X 0,Y 92.466,Z 759.102,A -85,B 0,C 180,E1 -27297.131,E2 -27297.131} C_VEL
LIN {X 0,Y 97.93,Z 752.846,A -85,B 0,C 180,E1 -27303.791,E2 -27303.791} C_VEL
LIN {X 0,Y 103.541,Z 745.99,A -85,B 0,C 180,E1 -27308.891,E2 -27308.891} C_VEL
LIN {X 0,Y 109.773,Z 737.388,A -85,B 0,C 180,E1 -27313.49,E2 -27313.49} C_VEL
LIN {X 0,Y 115.481,Z 728.568,A -85,B 0,C 180,E1 -27316.91,E2 -27316.91} C_VEL
LIN {X 0,Y 115.391,Z 727.148,A -85,B 0,C 180,E1 -27317.934,E2 -27317.934} C_VEL
LIN {X 0,Y 106.106,Z 728.335,A -85,B 0,C 180,E1 -27323.406,E2 -27323.406} C_VEL
LIN {X 0,Y 101.606,Z 729.261,A -85,B 0,C 180,E1 -27326.401,E2 -27326.401} C_VEL
LIN {X 0,Y 98.27,Z 729.098,A -85,B 0,C 180,E1 -27329.958,E2 -27329.958} C_VEL
LIN {X 0,Y 92.089,Z 729.67,A -85,B 0,C 180,E1 -27337.567,E2 -27337.567} C_VEL
LIN {X 0,Y 90.51,Z 728.981,A -85,B 0,C 180,E1 -27341.904,E2 -27341.904} C_VEL
LIN {X 0,Y 88.21,Z 729.715,A -85,B 0,C 180,E1 -27346.17,E2 -27346.17} C_VEL
LIN {X 0,Y 87.744,Z 728.953,A -85,B 0,C 180,E1 -27350.781,E2 -27350.781} C_VEL
LIN {X 0,Y 86.776,Z 729.414,A -85,B 0,C 180,E1 -27355.353,E2 -27355.353} C_VEL
LIN {X 0,Y 87.112,Z 728.927,A -85,B 0,C 180,E1 -27357.687,E2 -27357.687} C_VEL
LIN {X 0,Y 87.663,Z 728.438,A -85,B 0,C 180,E1 -27358.994,E2 -27358.994} C_VEL
LIN {X 0,Y 91.336,Z 734.401,A -85,B 0,C 180,E1 -27366.629,E2 -27366.629} C_VEL
LIN {X 0,Y 97.532,Z 739.815,A -85,B 0,C 180,E1 -27374.607,E2 -27374.607} C_VEL
LIN {X 0,Y 105.935,Z 743.837,A -85,B 0,C 180,E1 -27381.755,E2 -27381.755} C_VEL
LIN {X 0,Y 112.636,Z 745.697,A -85,B 0,C 180,E1 -27385.897,E2 -27385.897} C_VEL
LIN {X 0,Y 123.232,Z 747.138,A -85,B 0,C 180,E1 -27390.882,E2 -27390.882} C_VEL
LIN {X 0,Y 131.948,Z 747.274,A -85,B 0,C 180,E1 -27394.033,E2 -27394.033} C_VEL
LIN {X 0,Y 130.83,Z 747.566,A -85,B 0,C 180,E1 -27394.996,E2 -27394.996} C_VEL
LIN {X 0,Y 118.508,Z 748.829,A -85,B 0,C 180,E1 -27399.562,E2 -27399.562} C_VEL
LIN {X 0,Y 108.737,Z 748.788,A -85,B 0,C 180,E1 -27404.688,E2 -27404.688} C_VEL
LIN {X 0,Y 104.2,Z 748.375,A -85,B 0,C 180,E1 -27407.768,E2 -27407.768} C_VEL
LIN {X 0,Y 98.118,Z 755.525,A -85,B 0,C 180,E1 -27412.496,E2 -27412.496} C_VEL
LIN {X 0,Y 93.042,Z 761.416,A -85,B 0,C 180,E1 -27418.08,E2 -27418.08} C_VEL
LIN {X 0,Y 89.042,Z 766.055,A -85,B 0,C 180,E1 -27424.272,E2 -27424.272} C_VEL
LIN {X 0,Y 86.186,Z 769.577,A -85,B 0,C 180,E1 -27430.963,E2 -27430.963} C_VEL
LIN {X 0,Y 84.933,Z 771.354,A -85,B 0,C 180,E1 -27435.627,E2 -27435.627} C_VEL
LIN {X 0,Y 84.149,Z 772.691,A -85,B 0,C 180,E1 -27440.385,E2 -27440.385} C_VEL
LIN {X 0,Y 83.824,Z 773.632,A -85,B 0,C 180,E1 -27445.191,E2 -27445.191} C_VEL
LIN {X 0,Y 83.883,Z 774.172,A -85,B 0,C 180,E1 -27450,E2 -27450} C_VEL
LIN {X 0,Y 83.86,Z 774.256,A -85,B 0,C 180,E1 -27454.807,E2 -27454.807} C_VEL
LIN {X 0,Y 84.962,Z 773.247,A -85,B 0,C 180,E1 -27464.368,E2 -27464.368} C_VEL
LIN {X 0,Y 86.255,Z 772.143,A -85,B 0,C 180,E1 -27469.021,E2 -27469.021} C_VEL
LIN {X 0,Y 88.021,Z 770.59,A -85,B 0,C 180,E1 -27473.529,E2 -27473.529} C_VEL
LIN {X 0,Y 91.782,Z 767.478,A -85,B 0,C 180,E1 -27479.849,E2 -27479.849} C_VEL
LIN {X 0,Y 96.894,Z 762.96,A -85,B 0,C 180,E1 -27486.011,E2 -27486.011} C_VEL
LIN {X 0,Y 99.055,Z 760.449,A -85,B 0,C 180,E1 -27488.861,E2 -27488.861} C_VEL
LIN {X 0,Y 101.402,Z 755.938,A -85,B 0,C 180,E1 -27493.729,E2 -27493.729} C_VEL
LIN {X 0,Y 104.212,Z 750.865,A -85,B 0,C 180,E1 -27498.207,E2 -27498.207} C_VEL
LIN {X 0,Y 106.957,Z 747.378,A -85,B 0,C 180,E1 -27500.344,E2 -27500.344} C_VEL
LIN {X 0,Y 113.495,Z 739.587,A -85,B 0,C 180,E1 -27503.608,E2 -27503.608} C_VEL
LIN {X 0,Y 120.887,Z 729.227,A -85,B 0,C 180,E1 -27506.689,E2 -27506.689} C_VEL
LIN {X 0,Y 127.181,Z 718.694,A -85,B 0,C 180,E1 -27508.926,E2 -27508.926} C_VEL
LIN {X 0,Y 132.236,Z 708.502,A -85,B 0,C 180,E1 -27510.49,E2 -27510.49} C_VEL
LIN {X 0,Y 136.979,Z 696.311,A -85,B 0,C 180,E1 -27511.863,E2 -27511.863} C_VEL
LIN {X 0,Y 140.713,Z 683.597,A -85,B 0,C 180,E1 -27512.827,E2 -27512.827} C_VEL
LIN {X 0,Y 143.156,Z 670.953,A -85,B 0,C 180,E1 -27513.477,E2 -27513.477} C_VEL
LIN {X 0,Y 146.898,Z 634.053,A -85,B 0,C 180,E1 -27514.709,E2 -27514.709} C_VEL
LIN {X 0,Y 144.528,Z 628.34,A -85,B 0,C 180,E1 -27517.616,E2 -27517.616} C_VEL
LIN {X 0,Y 142.252,Z 623.027,A -85,B 0,C 180,E1 -27520.902,E2 -27520.902} C_VEL
LIN {X 0,Y 140.246,Z 618.914,A -85,B 0,C 180,E1 -27524.375,E2 -27524.375} C_VEL
LIN {X 0,Y 138.812,Z 615.955,A -85,B 0,C 180,E1 -27527.557,E2 -27527.557} C_VEL
LIN {X 0,Y 137.29,Z 612.576,A -85,B 0,C 180,E1 -27532.648,E2 -27532.648} C_VEL
LIN {X 0,Y 136.603,Z 611.103,A -85,B 0,C 180,E1 -27538.914,E2 -27538.914} C_VEL
LIN {X 0,Y 136.659,Z 611.319,A -85,B 0,C 180,E1 -27541.106,E2 -27541.106} C_VEL
LIN {X 0,Y 137.438,Z 612.984,A -85,B 0,C 180,E1 -27546.239,E2 -27546.239} C_VEL
LIN {X 0,Y 138.882,Z 616.074,A -85,B 0,C 180,E1 -27550.801,E2 -27550.801} C_VEL
LIN {X 0,Y 140.714,Z 620.1,A -85,B 0,C 180,E1 -27554.739,E2 -27554.739} C_VEL
LIN {X 0,Y 142.295,Z 623.574,A -85,B 0,C 180,E1 -27557.424,E2 -27557.424} C_VEL
LIN {X 0,Y 144.51,Z 629.029,A -85,B 0,C 180,E1 -27560.647,E2 -27560.647} C_VEL
LIN {X 0,Y 146.927,Z 635.818,A -85,B 0,C 180,E1 -27563.71,E2 -27563.71} C_VEL
LIN {X 0,Y 143.561,Z 668.161,A -85,B 0,C 180,E1 -27564.773,E2 -27564.773} C_VEL
LIN {X 0,Y 140.906,Z 681.483,A -85,B 0,C 180,E1 -27565.53,E2 -27565.53} C_VEL
LIN {X 0,Y 137.092,Z 694.357,A -85,B 0,C 180,E1 -27566.631,E2 -27566.631} C_VEL
LIN {X 0,Y 132.479,Z 706.111,A -85,B 0,C 180,E1 -27568.123,E2 -27568.123} C_VEL
LIN {X 0,Y 127.32,Z 716.633,A -85,B 0,C 180,E1 -27569.965,E2 -27569.965} C_VEL
LIN {X 0,Y 120.812,Z 727.475,A -85,B 0,C 180,E1 -27572.49,E2 -27572.49} C_VEL
LIN {X 0,Y 114.182,Z 736.576,A -85,B 0,C 180,E1 -27575.36,E2 -27575.36} C_VEL
LIN {X 0,Y 106.684,Z 745.38,A -85,B 0,C 180,E1 -27579.283,E2 -27579.283} C_VEL
LIN {X 0,Y 99.726,Z 752.461,A -85,B 0,C 180,E1 -27583.753,E2 -27583.753} C_VEL
LIN {X 0,Y 93.326,Z 758.272,A -85,B 0,C 180,E1 -27589.124,E2 -27589.124} C_VEL
LIN {X 0,Y 87.4,Z 763.084,A -85,B 0,C 180,E1 -27595.746,E2 -27595.746} C_VEL
LIN {X 0,Y 84.33,Z 765.305,A -85,B 0,C 180,E1 -27599.998,E2 -27599.998} C_VEL
LIN {X 0,Y 81.761,Z 767.069,A -85,B 0,C 180,E1 -27604.546,E2 -27604.546} C_VEL
LIN {X 0,Y 79.788,Z 768.384,A -85,B 0,C 180,E1 -27609.37,E2 -27609.37} C_VEL
LIN {X 0,Y 78.29,Z 769.309,A -85,B 0,C 180,E1 -27614.377,E2 -27614.377} C_VEL
LIN {X 0,Y 77.294,Z 769.848,A -85,B 0,C 180,E1 -27619.523,E2 -27619.523} C_VEL
LIN {X 0,Y 76.803,Z 769.955,A -85,B 0,C 180,E1 -27624.75,E2 -27624.75} C_VEL
LIN {X 0,Y 76.787,Z 769.671,A -85,B 0,C 180,E1 -27630,E2 -27630} C_VEL
LIN {X 0,Y 77.217,Z 769.009,A -85,B 0,C 180,E1 -27635.222,E2 -27635.222} C_VEL
LIN {X 0,Y 78.048,Z 767.957,A -85,B 0,C 180,E1 -27640.375,E2 -27640.375} C_VEL
LIN {X 0,Y 79.326,Z 766.457,A -85,B 0,C 180,E1 -27645.413,E2 -27645.413} C_VEL
LIN {X 0,Y 82.201,Z 763.43,A -85,B 0,C 180,E1 -27652.627,E2 -27652.627} C_VEL
LIN {X 0,Y 86.222,Z 759.347,A -85,B 0,C 180,E1 -27659.278,E2 -27659.278} C_VEL
LIN {X 0,Y 92.123,Z 753.104,A -85,B 0,C 180,E1 -27666.244,E2 -27666.244} C_VEL
LIN {X 0,Y 98.129,Z 746.269,A -85,B 0,C 180,E1 -27671.488,E2 -27671.488} C_VEL
LIN {X 0,Y 104.753,Z 737.685,A -85,B 0,C 180,E1 -27676.155,E2 -27676.155} C_VEL
LIN {X 0,Y 107.016,Z 734.512,A -85,B 0,C 180,E1 -27677.519,E2 -27677.519} C_VEL
LIN {X 0,Y 107.575,Z 732.913,A -85,B 0,C 180,E1 -27678.503,E2 -27678.503} C_VEL
LIN {X 0,Y 97.575,Z 734.389,A -85,B 0,C 180,E1 -27684.814,E2 -27684.814} C_VEL
LIN {X 0,Y 94.075,Z 734.256,A -85,B 0,C 180,E1 -27688.469,E2 -27688.469} C_VEL
LIN {X 0,Y 87.589,Z 734.818,A -85,B 0,C 180,E1 -27696.346,E2 -27696.346} C_VEL
LIN {X 0,Y 85.87,Z 734.217,A -85,B 0,C 180,E1 -27700.889,E2 -27700.889} C_VEL
LIN {X 0,Y 83.487,Z 734.877,A -85,B 0,C 180,E1 -27705.371,E2 -27705.371} C_VEL
LIN {X 0,Y 82.927,Z 734.235,A -85,B 0,C 180,E1 -27710.24,E2 -27710.24} C_VEL
LIN {X 0,Y 81.97,Z 734.597,A -85,B 0,C 180,E1 -27715.08,E2 -27715.08} C_VEL
LIN {X 0,Y 82.633,Z 733.933,A -85,B 0,C 180,E1 -27719.999,E2 -27719.999} C_VEL
LIN {X 0,Y 83.086,Z 734.078,A -85,B 0,C 180,E1 -27724.851,E2 -27724.851} C_VEL
LIN {X 0,Y 84.486,Z 733.302,A -85,B 0,C 180,E1 -27727.837,E2 -27727.837} C_VEL
LIN {X 0,Y 84.884,Z 733.167,A -85,B 0,C 180,E1 -27728.368,E2 -27728.368} C_VEL
LIN {X 0,Y 90.502,Z 738.355,A -85,B 0,C 180,E1 -27735.77,E2 -27735.77} C_VEL
LIN {X 0,Y 96.549,Z 741.877,A -85,B 0,C 180,E1 -27741.343,E2 -27741.343} C_VEL
LIN {X 0,Y 106.05,Z 745.346,A -85,B 0,C 180,E1 -27747.638,E2 -27747.638} C_VEL
LIN {X 0,Y 117.029,Z 747.459,A -85,B 0,C 180,E1 -27752.783,E2 -27752.783} C_VEL
LIN {X 0,Y 119.687,Z 747.901,A -85,B 0,C 180,E1 -27754.709,E2 -27754.709} C_VEL
LIN {X 0,Y 108.885,Z 747.985,A -85,B 0,C 180,E1 -27759.238,E2 -27759.238} C_VEL
LIN {X 0,Y 99.846,Z 747.244,A -85,B 0,C 180,E1 -27764.548,E2 -27764.548} C_VEL
LIN {X 0,Y 93.76,Z 753.956,A -85,B 0,C 180,E1 -27768.763,E2 -27768.763} C_VEL
LIN {X 0,Y 88.804,Z 759.362,A -85,B 0,C 180,E1 -27773.592,E2 -27773.592} C_VEL
LIN {X 0,Y 84.043,Z 764.395,A -85,B 0,C 180,E1 -27779.885,E2 -27779.885} C_VEL
LIN {X 0,Y 80.356,Z 768.283,A -85,B 0,C 180,E1 -27786.824,E2 -27786.824} C_VEL
LIN {X 0,Y 78.036,Z 771.138,A -85,B 0,C 180,E1 -27794.325,E2 -27794.325} C_VEL
LIN {X 0,Y 77.132,Z 772.481,A -85,B 0,C 180,E1 -27799.5,E2 -27799.5} C_VEL
LIN {X 0,Y 76.752,Z 773.428,A -85,B 0,C 180,E1 -27804.746,E2 -27804.746} C_VEL
LIN {X 0,Y 76.781,Z 773.975,A -85,B 0,C 180,E1 -27810,E2 -27810} C_VEL
LIN {X 0,Y 76.779,Z 774.067,A -85,B 0,C 180,E1 -27815.252,E2 -27815.252} C_VEL
LIN {X 0,Y 78.066,Z 773.069,A -85,B 0,C 180,E1 -27825.669,E2 -27825.669} C_VEL
LIN {X 0,Y 79.555,Z 771.975,A -85,B 0,C 180,E1 -27830.693,E2 -27830.693} C_VEL
LIN {X 0,Y 81.526,Z 770.428,A -85,B 0,C 180,E1 -27835.532,E2 -27835.532} C_VEL
LIN {X 0,Y 85.675,Z 767.329,A -85,B 0,C 180,E1 -27842.221,E2 -27842.221} C_VEL
LIN {X 0,Y 90.851,Z 763.154,A -85,B 0,C 180,E1 -27848.257,E2 -27848.257} C_VEL
LIN {X 0,Y 97.727,Z 756.919,A -85,B 0,C 180,E1 -27854.375,E2 -27854.375} C_VEL
LIN {X 0,Y 104.666,Z 749.88,A -85,B 0,C 180,E1 -27859.059,E2 -27859.059} C_VEL
LIN {X 0,Y 106.957,Z 747.378,A -85,B 0,C 180,E1 -27860.344,E2 -27860.344} C_VEL
LIN {X 0,Y 109.786,Z 743.74,A -85,B 0,C 180,E1 -27862.302,E2 -27862.302} C_VEL
LIN {X 0,Y 113.234,Z 737.439,A -85,B 0,C 180,E1 -27865.817,E2 -27865.817} C_VEL
LIN {X 0,Y 116.615,Z 730.576,A -85,B 0,C 180,E1 -27868.965,E2 -27868.965} C_VEL
LIN {X 0,Y 119.213,Z 726.056,A -85,B 0,C 180,E1 -27870.322,E2 -27870.322} C_VEL
LIN {X 0,Y 125.885,Z 714.58,A -85,B 0,C 180,E1 -27872.407,E2 -27872.407} C_VEL
LIN {X 0,Y 131.149,Z 703.397,A -85,B 0,C 180,E1 -27873.841,E2 -27873.841} C_VEL
LIN {X 0,Y 135.696,Z 690.672,A -85,B 0,C 180,E1 -27875.003,E2 -27875.003} C_VEL
LIN {X 0,Y 139.069,Z 677.488,A -85,B 0,C 180,E1 -27875.808,E2 -27875.808} C_VEL
LIN {X 0,Y 141.063,Z 664.041,A -85,B 0,C 180,E1 -27876.361,E2 -27876.361} C_VEL
LIN {X 0,Y 143.721,Z 637.462,A -85,B 0,C 180,E1 -27877.219,E2 -27877.219} C_VEL
LIN {X 0,Y 140.889,Z 630.082,A -85,B 0,C 180,E1 -27881.469,E2 -27881.469} C_VEL
LIN {X 0,Y 138.822,Z 625.462,A -85,B 0,C 180,E1 -27885.338,E2 -27885.338} C_VEL
LIN {X 0,Y 137.51,Z 622.527,A -85,B 0,C 180,E1 -27888.578,E2 -27888.578} C_VEL
LIN {X 0,Y 136.34,Z 619.585,A -85,B 0,C 180,E1 -27892.969,E2 -27892.969} C_VEL
LIN {X 0,Y 135.736,Z 618.166,A -85,B 0,C 180,E1 -27898.907,E2 -27898.907} C_VEL
LIN {X 0,Y 135.81,Z 618.513,A -85,B 0,C 180,E1 -27901.483,E2 -27901.483} C_VEL
LIN {X 0,Y 136.411,Z 619.885,A -85,B 0,C 180,E1 -27905.637,E2 -27905.637} C_VEL
LIN {X 0,Y 137.686,Z 622.923,A -85,B 0,C 180,E1 -27910.106,E2 -27910.106} C_VEL
LIN {X 0,Y 139.203,Z 626.53,A -85,B 0,C 180,E1 -27913.69,E2 -27913.69} C_VEL
LIN {X 0,Y 140.731,Z 630.274,A -85,B 0,C 180,E1 -27916.548,E2 -27916.548} C_VEL
LIN {X 0,Y 142.769,Z 635.89,A -85,B 0,C 180,E1 -27919.782,E2 -27919.782} C_VEL
LIN {X 0,Y 143.772,Z 638.984,A -85,B 0,C 180,E1 -27921.221,E2 -27921.221} C_VEL
LIN {X 0,Y 140.491,Z 669.131,A -85,B 0,C 180,E1 -27922.207,E2 -27922.207} C_VEL
LIN {X 0,Y 137.658,Z 682.513,A -85,B 0,C 180,E1 -27922.953,E2 -27922.953} C_VEL
LIN {X 0,Y 133.685,Z 695.29,A -85,B 0,C 180,E1 -27924.019,E2 -27924.019} C_VEL
LIN {X 0,Y 128.54,Z 707.61,A -85,B 0,C 180,E1 -27925.561,E2 -27925.561} C_VEL
LIN {X 0,Y 122.757,Z 718.71,A -85,B 0,C 180,E1 -27927.53,E2 -27927.53} C_VEL
LIN {X 0,Y 117.141,Z 727.511,A -85,B 0,C 180,E1 -27929.551,E2 -27929.551} C_VEL
LIN {X 0,Y 110.221,Z 736.649,A -85,B 0,C 180,E1 -27932.346,E2 -27932.346} C_VEL
LIN {X 0,Y 102.326,Z 745.474,A -85,B 0,C 180,E1 -27936.196,E2 -27936.196} C_VEL
LIN {X 0,Y 94.926,Z 752.574,A -85,B 0,C 180,E1 -27940.637,E2 -27940.637} C_VEL
LIN {X 0,Y 87.642,Z 758.716,A -85,B 0,C 180,E1 -27946.446,E2 -27946.446} C_VEL
LIN {X 0,Y 81.613,Z 763.232,A -85,B 0,C 180,E1 -27952.931,E2 -27952.931} C_VEL
LIN {X 0,Y 78.258,Z 765.458,A -85,B 0,C 180,E1 -27957.397,E2 -27957.397} C_VEL
LIN {X 0,Y 75.38,Z 767.236,A -85,B 0,C 180,E1 -27962.215,E2 -27962.215} C_VEL
LIN {X 0,Y 71.46,Z 769.486,A -85,B 0,C 180,E1 -27972.84,E2 -27972.84} C_VEL
LIN {X 0,Y 70.321,Z 770.032,A -85,B 0,C 180,E1 -27978.47,E2 -27978.47} C_VEL
LIN {X 0,Y 69.747,Z 770.149,A -85,B 0,C 180,E1 -27984.217,E2 -27984.217} C_VEL
LIN {X 0,Y 69.708,Z 769.87,A -85,B 0,C 180,E1 -27990,E2 -27990} C_VEL
LIN {X 0,Y 70.17,Z 769.213,A -85,B 0,C 180,E1 -27995.748,E2 -27995.748} C_VEL
LIN {X 0,Y 71.101,Z 768.17,A -85,B 0,C 180,E1 -28001.402,E2 -28001.402} C_VEL
LIN {X 0,Y 72.522,Z 766.678,A -85,B 0,C 180,E1 -28006.901,E2 -28006.901} C_VEL
LIN {X 0,Y 75.7,Z 763.663,A -85,B 0,C 180,E1 -28014.694,E2 -28014.694} C_VEL
LIN {X 0,Y 80.122,Z 759.592,A -85,B 0,C 180,E1 -28021.755,E2 -28021.755} C_VEL
LIN {X 0,Y 86.51,Z 753.362,A -85,B 0,C 180,E1 -28029.02,E2 -28029.02} C_VEL
LIN {X 0,Y 92.937,Z 746.547,A -85,B 0,C 180,E1 -28034.385,E2 -28034.385} C_VEL
LIN {X 0,Y 98.151,Z 740.31,A -85,B 0,C 180,E1 -28037.986,E2 -28037.986} C_VEL
LIN {X 0,Y 99.036,Z 738.366,A -85,B 0,C 180,E1 -28039.382,E2 -28039.382} C_VEL
LIN {X 0,Y 93.405,Z 739.249,A -85,B 0,C 180,E1 -28042.99,E2 -28042.99} C_VEL
LIN {X 0,Y 89.721,Z 739.14,A -85,B 0,C 180,E1 -28046.747,E2 -28046.747} C_VEL
LIN {X 0,Y 82.893,Z 739.688,A -85,B 0,C 180,E1 -28054.916,E2 -28054.916} C_VEL
LIN {X 0,Y 80.988,Z 739.183,A -85,B 0,C 180,E1 -28059.688,E2 -28059.688} C_VEL
LIN {X 0,Y 78.518,Z 739.767,A -85,B 0,C 180,E1 -28064.422,E2 -28064.422} C_VEL
LIN {X 0,Y 77.843,Z 739.213,A -85,B 0,C 180,E1 -28069.596,E2 -28069.596} C_VEL
LIN {X 0,Y 76.887,Z 739.505,A -85,B 0,C 180,E1 -28074.754,E2 -28074.754} C_VEL
LIN {X 0,Y 77.502,Z 738.943,A -85,B 0,C 180,E1 -28079.999,E2 -28079.999} C_VEL
LIN {X 0,Y 78.031,Z 739.042,A -85,B 0,C 180,E1 -28085.166,E2 -28085.166} C_VEL
LIN {X 0,Y 80.025,Z 738.359,A -85,B 0,C 180,E1 -28090.115,E2 -28090.115} C_VEL
LIN {X 0,Y 81.897,Z 738.322,A -85,B 0,C 180,E1 -28094.917,E2 -28094.917} C_VEL
LIN {X 0,Y 84.769,Z 737.491,A -85,B 0,C 180,E1 -28098.425,E2 -28098.425} C_VEL
LIN {X 0,Y 94.016,Z 742.616,A -85,B 0,C 180,E1 -28106.232,E2 -28106.232} C_VEL
LIN {X 0,Y 104.998,Z 746.217,A -85,B 0,C 180,E1 -28112.375,E2 -28112.375} C_VEL
LIN {X 0,Y 108.342,Z 746.954,A -85,B 0,C 180,E1 -28113.849,E2 -28113.849} C_VEL
LIN {X 0,Y 106.594,Z 747.023,A -85,B 0,C 180,E1 -28115.342,E2 -28115.342} C_VEL
LIN {X 0,Y 95.994,Z 745.893,A -85,B 0,C 180,E1 -28120.975,E2 -28120.975} C_VEL
LIN {X 0,Y 89.48,Z 752.733,A -85,B 0,C 180,E1 -28125.019,E2 -28125.019} C_VEL
LIN {X 0,Y 83.186,Z 759.111,A -85,B 0,C 180,E1 -28130.682,E2 -28130.682} C_VEL
LIN {X 0,Y 77.961,Z 764.157,A -85,B 0,C 180,E1 -28137.257,E2 -28137.257} C_VEL
LIN {X 0,Y 73.843,Z 768.056,A -85,B 0,C 180,E1 -28144.642,E2 -28144.642} C_VEL
LIN {X 0,Y 71.198,Z 770.922,A -85,B 0,C 180,E1 -28152.775,E2 -28152.775} C_VEL
LIN {X 0,Y 70.148,Z 772.271,A -85,B 0,C 180,E1 -28158.441,E2 -28158.441} C_VEL
LIN {X 0,Y 69.662,Z 773.223,A -85,B 0,C 180,E1 -28164.21,E2 -28164.21} C_VEL
LIN {X 0,Y 69.701,Z 773.779,A -85,B 0,C 180,E1 -28170,E2 -28170} C_VEL
LIN {X 0,Y 69.702,Z 773.878,A -85,B 0,C 180,E1 -28175.787,E2 -28175.787} C_VEL
LIN {X 0,Y 71.231,Z 772.891,A -85,B 0,C 180,E1 -28187.217,E2 -28187.217} C_VEL
LIN {X 0,Y 72.922,Z 771.806,A -85,B 0,C 180,E1 -28192.675,E2 -28192.675} C_VEL
LIN {X 0,Y 75.151,Z 770.266,A -85,B 0,C 180,E1 -28197.878,E2 -28197.878} C_VEL
LIN {X 0,Y 79.738,Z 767.179,A -85,B 0,C 180,E1 -28204.952,E2 -28204.952} C_VEL
LIN {X 0,Y 85.359,Z 763.032,A -85,B 0,C 180,E1 -28211.198,E2 -28211.198} C_VEL
LIN {X 0,Y 92.761,Z 756.797,A -85,B 0,C 180,E1 -28217.459,E2 -28217.459} C_VEL
LIN {X 0,Y 100.154,Z 749.781,A -85,B 0,C 180,E1 -28222.131,E2 -28222.131} C_VEL
LIN {X 0,Y 108.065,Z 741.119,A -85,B 0,C 180,E1 -28226.014,E2 -28226.014} C_VEL
LIN {X 0,Y 115.729,Z 731.277,A -85,B 0,C 180,E1 -28229.066,E2 -28229.066} C_VEL
LIN {X 0,Y 119.213,Z 726.056,A -85,B 0,C 180,E1 -28230.322,E2 -28230.322} C_VEL
LIN {X 0,Y 121.736,Z 721.402,A -85,B 0,C 180,E1 -28231.566,E2 -28231.566} C_VEL
LIN {X 0,Y 125.881,Z 710.39,A -85,B 0,C 180,E1 -28234.978,E2 -28234.978} C_VEL
LIN {X 0,Y 128.199,Z 703.704,A -85,B 0,C 180,E1 -28236.532,E2 -28236.532} C_VEL
LIN {X 0,Y 129.552,Z 700.109,A -85,B 0,C 180,E1 -28237.01,E2 -28237.01} C_VEL
LIN {X 0,Y 133.832,Z 687.732,A -85,B 0,C 180,E1 -28237.986,E2 -28237.986} C_VEL
LIN {X 0,Y 136.746,Z 675.685,A -85,B 0,C 180,E1 -28238.625,E2 -28238.625} C_VEL
LIN {X 0,Y 138.755,Z 661.482,A -85,B 0,C 180,E1 -28239.138,E2 -28239.138} C_VEL
LIN {X 0,Y 140.873,Z 641.114,A -85,B 0,C 180,E1 -28239.753,E2 -28239.753} C_VEL
LIN {X 0,Y 138.596,Z 634.823,A -85,B 0,C 180,E1 -28243.806,E2 -28243.806} C_VEL
LIN {X 0,Y 136.978,Z 630.872,A -85,B 0,C 180,E1 -28247.484,E2 -28247.484} C_VEL
LIN {X 0,Y 136.198,Z 629.012,A -85,B 0,C 180,E1 -28249.783,E2 -28249.783} C_VEL
LIN {X 0,Y 135.259,Z 626.34,A -85,B 0,C 180,E1 -28254.036,E2 -28254.036} C_VEL
LIN {X 0,Y 134.871,Z 625.206,A -85,B 0,C 180,E1 -28258.9,E2 -28258.9} C_VEL
LIN {X 0,Y 135.022,Z 625.821,A -85,B 0,C 180,E1 -28262.425,E2 -28262.425} C_VEL
LIN {X 0,Y 135.419,Z 626.822,A -85,B 0,C 180,E1 -28265.118,E2 -28265.118} C_VEL
LIN {X 0,Y 136.47,Z 629.623,A -85,B 0,C 180,E1 -28269.262,E2 -28269.262} C_VEL
LIN {X 0,Y 137.774,Z 633.098,A -85,B 0,C 180,E1 -28272.709,E2 -28272.709} C_VEL
LIN {X 0,Y 139.062,Z 636.572,A -85,B 0,C 180,E1 -28275.387,E2 -28275.387} C_VEL
LIN {X 0,Y 140.665,Z 641.593,A -85,B 0,C 180,E1 -28278.269,E2 -28278.269} C_VEL
LIN {X 0,Y 140.895,Z 642.409,A -85,B 0,C 180,E1 -28278.658,E2 -28278.658} C_VEL
LIN {X 0,Y 137.834,Z 669.382,A -85,B 0,C 180,E1 -28279.507,E2 -28279.507} C_VEL
LIN {X 0,Y 134.988,Z 682.485,A -85,B 0,C 180,E1 -28280.193,E2 -28280.193} C_VEL
LIN {X 0,Y 130.959,Z 695.165,A -85,B 0,C 180,E1 -28281.185,E2 -28281.185} C_VEL
LIN {X 0,Y 126.401,Z 706.028,A -85,B 0,C 180,E1 -28282.431,E2 -28282.431} C_VEL
LIN {X 0,Y 120.451,Z 717.278,A -85,B 0,C 180,E1 -28284.212,E2 -28284.212} C_VEL
LIN {X 0,Y 113.81,Z 727.546,A -85,B 0,C 180,E1 -28286.442,E2 -28286.442} C_VEL
LIN {X 0,Y 106.583,Z 736.722,A -85,B 0,C 180,E1 -28289.112,E2 -28289.112} C_VEL
LIN {X 0,Y 98.294,Z 745.567,A -85,B 0,C 180,E1 -28292.85,E2 -28292.85} C_VEL
LIN {X 0,Y 90.455,Z 752.686,A -85,B 0,C 180,E1 -28297.216,E2 -28297.216} C_VEL
LIN {X 0,Y 83.096,Z 758.491,A -85,B 0,C 180,E1 -28302.582,E2 -28302.582} C_VEL
LIN {X 0,Y 76.034,Z 763.38,A -85,B 0,C 180,E1 -28309.683,E2 -28309.683} C_VEL
LIN {X 0,Y 72.372,Z 765.612,A -85,B 0,C 180,E1 -28314.363,E2 -28314.363} C_VEL
LIN {X 0,Y 69.15,Z 767.402,A -85,B 0,C 180,E1 -28319.459,E2 -28319.459} C_VEL
LIN {X 0,Y 64.701,Z 769.664,A -85,B 0,C 180,E1 -28330.982,E2 -28330.982} C_VEL
LIN {X 0,Y 63.361,Z 770.216,A -85,B 0,C 180,E1 -28337.183,E2 -28337.183} C_VEL
LIN {X 0,Y 62.674,Z 770.343,A -85,B 0,C 180,E1 -28343.562,E2 -28343.562} C_VEL
LIN {X 0,Y 62.62,Z 770.069,A -85,B 0,C 180,E1 -28350,E2 -28350} C_VEL
LIN {X 0,Y 63.117,Z 769.418,A -85,B 0,C 180,E1 -28356.393,E2 -28356.393} C_VEL
LIN {X 0,Y 64.171,Z 768.382,A -85,B 0,C 180,E1 -28362.652,E2 -28362.652} C_VEL
LIN {X 0,Y 65.771,Z 766.9,A -85,B 0,C 180,E1 -28368.697,E2 -28368.697} C_VEL
LIN {X 0,Y 69.324,Z 763.896,A -85,B 0,C 180,E1 -28377.142,E2 -28377.142} C_VEL
LIN {X 0,Y 74.185,Z 759.837,A -85,B 0,C 180,E1 -28384.639,E2 -28384.639} C_VEL
LIN {X 0,Y 81.131,Z 753.62,A -85,B 0,C 180,E1 -28392.17,E2 -28392.17} C_VEL
LIN {X 0,Y 88.013,Z 746.824,A -85,B 0,C 180,E1 -28397.613,E2 -28397.613} C_VEL
LIN {X 0,Y 89.187,Z 745.507,A -85,B 0,C 180,E1 -28398.468,E2 -28398.468} C_VEL
LIN {X 0,Y 90.103,Z 743.699,A -85,B 0,C 180,E1 -28400.196,E2 -28400.196} C_VEL
LIN {X 0,Y 81.431,Z 743.973,A -85,B 0,C 180,E1 -28408.811,E2 -28408.811} C_VEL
LIN {X 0,Y 78.024,Z 744.252,A -85,B 0,C 180,E1 -28413.231,E2 -28413.231} C_VEL
LIN {X 0,Y 75.915,Z 743.844,A -85,B 0,C 180,E1 -28418.264,E2 -28418.264} C_VEL
LIN {X 0,Y 73.145,Z 744.357,A -85,B 0,C 180,E1 -28423.904,E2 -28423.904} C_VEL
LIN {X 0,Y 72.513,Z 743.897,A -85,B 0,C 180,E1 -28428.822,E2 -28428.822} C_VEL
LIN {X 0,Y 71.535,Z 744.14,A -85,B 0,C 180,E1 -28434.36,E2 -28434.36} C_VEL
LIN {X 0,Y 72.086,Z 743.677,A -85,B 0,C 180,E1 -28439.999,E2 -28439.999} C_VEL
LIN {X 0,Y 72.72,Z 743.716,A -85,B 0,C 180,E1 -28445.545,E2 -28445.545} C_VEL
LIN {X 0,Y 74.729,Z 743.153,A -85,B 0,C 180,E1 -28450.84,E2 -28450.84} C_VEL
LIN {X 0,Y 76.814,Z 743.046,A -85,B 0,C 180,E1 -28455.93,E2 -28455.93} C_VEL
LIN {X 0,Y 80.195,Z 742.288,A -85,B 0,C 180,E1 -28460.52,E2 -28460.52} C_VEL
LIN {X 0,Y 83.358,Z 742.151,A -85,B 0,C 180,E1 -28464.932,E2 -28464.932} C_VEL
LIN {X 0,Y 87.344,Z 741.176,A -85,B 0,C 180,E1 -28468.21,E2 -28468.21} C_VEL
LIN {X 0,Y 96.952,Z 744.965,A -85,B 0,C 180,E1 -28473.785,E2 -28473.785} C_VEL
LIN {X 0,Y 95.158,Z 744.88,A -85,B 0,C 180,E1 -28475.669,E2 -28475.669} C_VEL
LIN {X 0,Y 92.548,Z 744.508,A -85,B 0,C 180,E1 -28477.123,E2 -28477.123} C_VEL
LIN {X 0,Y 85.857,Z 751.243,A -85,B 0,C 180,E1 -28480.786,E2 -28480.786} C_VEL
LIN {X 0,Y 79.956,Z 756.865,A -85,B 0,C 180,E1 -28485.318,E2 -28485.318} C_VEL
LIN {X 0,Y 73.828,Z 762.344,A -85,B 0,C 180,E1 -28491.775,E2 -28491.775} C_VEL
LIN {X 0,Y 68.841,Z 766.629,A -85,B 0,C 180,E1 -28499.307,E2 -28499.307} C_VEL
LIN {X 0,Y 66.273,Z 768.895,A -85,B 0,C 180,E1 -28504.902,E2 -28504.902} C_VEL
LIN {X 0,Y 64.429,Z 770.706,A -85,B 0,C 180,E1 -28510.899,E2 -28510.899} C_VEL
LIN {X 0,Y 63.181,Z 772.061,A -85,B 0,C 180,E1 -28517.146,E2 -28517.146} C_VEL
LIN {X 0,Y 62.587,Z 773.018,A -85,B 0,C 180,E1 -28523.553,E2 -28523.553} C_VEL
LIN {X 0,Y 62.611,Z 773.582,A -85,B 0,C 180,E1 -28530,E2 -28530} C_VEL
LIN {X 0,Y 62.619,Z 773.689,A -85,B 0,C 180,E1 -28536.444,E2 -28536.444} C_VEL
LIN {X 0,Y 64.466,Z 772.713,A -85,B 0,C 180,E1 -28549.09,E2 -28549.09} C_VEL
LIN {X 0,Y 66.38,Z 771.636,A -85,B 0,C 180,E1 -28555.055,E2 -28555.055} C_VEL
LIN {X 0,Y 68.93,Z 770.105,A -85,B 0,C 180,E1 -28560.649,E2 -28560.649} C_VEL
LIN {X 0,Y 74.011,Z 767.03,A -85,B 0,C 180,E1 -28568.113,E2 -28568.113} C_VEL
LIN {X 0,Y 81.65,Z 761.785,A -85,B 0,C 180,E1 -28575.918,E2 -28575.918} C_VEL
LIN {X 0,Y 89.458,Z 755.534,A -85,B 0,C 180,E1 -28581.776,E2 -28581.776} C_VEL
LIN {X 0,Y 97.307,Z 748.346,A -85,B 0,C 180,E1 -28586.157,E2 -28586.157} C_VEL
LIN {X 0,Y 105.692,Z 739.435,A -85,B 0,C 180,E1 -28589.816,E2 -28589.816} C_VEL
LIN {X 0,Y 113.714,Z 729.146,A -85,B 0,C 180,E1 -28592.674,E2 -28592.674} C_VEL
LIN {X 0,Y 120.479,Z 718.678,A -85,B 0,C 180,E1 -28594.709,E2 -28594.709} C_VEL
LIN {X 0,Y 125.861,Z 708.582,A -85,B 0,C 180,E1 -28596.114,E2 -28596.114} C_VEL
LIN {X 0,Y 129.552,Z 700.109,A -85,B 0,C 180,E1 -28597.01,E2 -28597.01} C_VEL
LIN {X 0,Y 131.342,Z 694.732,A -85,B 0,C 180,E1 -28597.743,E2 -28597.743} C_VEL
LIN {X 0,Y 133.126,Z 685.856,A -85,B 0,C 180,E1 -28599.489,E2 -28599.489} C_VEL
LIN {X 0,Y 134.445,Z 676.764,A -85,B 0,C 180,E1 -28601.095,E2 -28601.095} C_VEL
LIN {X 0,Y 135.279,Z 671.047,A -85,B 0,C 180,E1 -28601.618,E2 -28601.618} C_VEL
LIN {X 0,Y 138.245,Z 644.908,A -85,B 0,C 180,E1 -28602.453,E2 -28602.453} C_VEL
LIN {X 0,Y 136.924,Z 640.83,A -85,B 0,C 180,E1 -28605.263,E2 -28605.263} C_VEL
LIN {X 0,Y 135.374,Z 636.432,A -85,B 0,C 180,E1 -28609.532,E2 -28609.532} C_VEL
LIN {X 0,Y 134.277,Z 633.192,A -85,B 0,C 180,E1 -28614.745,E2 -28614.745} C_VEL
LIN {X 0,Y 134.019,Z 632.271,A -85,B 0,C 180,E1 -28620.001,E2 -28620.001} C_VEL
LIN {X 0,Y 134.425,Z 633.694,A -85,B 0,C 180,E1 -28624.499,E2 -28624.499} C_VEL
LIN {X 0,Y 135.393,Z 636.633,A -85,B 0,C 180,E1 -28628.771,E2 -28628.771} C_VEL
LIN {X 0,Y 136.919,Z 641.123,A -85,B 0,C 180,E1 -28632.981,E2 -28632.981} C_VEL
LIN {X 0,Y 138.315,Z 645.885,A -85,B 0,C 180,E1 -28636.007,E2 -28636.007} C_VEL
LIN {X 0,Y 135.461,Z 669.785,A -85,B 0,C 180,E1 -28636.708,E2 -28636.708} C_VEL
LIN {X 0,Y 132.532,Z 682.859,A -85,B 0,C 180,E1 -28637.352,E2 -28637.352} C_VEL
LIN {X 0,Y 128.563,Z 695.028,A -85,B 0,C 180,E1 -28638.233,E2 -28638.233} C_VEL
LIN {X 0,Y 123.86,Z 705.985,A -85,B 0,C 180,E1 -28639.385,E2 -28639.385} C_VEL
LIN {X 0,Y 118.32,Z 716.281,A -85,B 0,C 180,E1 -28640.88,E2 -28640.88} C_VEL
LIN {X 0,Y 111.599,Z 726.533,A -85,B 0,C 180,E1 -28642.929,E2 -28642.929} C_VEL
LIN {X 0,Y 104.786,Z 735.078,A -85,B 0,C 180,E1 -28645.12,E2 -28645.12} C_VEL
LIN {X 0,Y 97.489,Z 742.928,A -85,B 0,C 180,E1 -28647.984,E2 -28647.984} C_VEL
LIN {X 0,Y 89.05,Z 750.599,A -85,B 0,C 180,E1 -28651.963,E2 -28651.963} C_VEL
LIN {X 0,Y 82.397,Z 755.809,A -85,B 0,C 180,E1 -28655.877,E2 -28655.877} C_VEL
LIN {X 0,Y 75.143,Z 760.845,A -85,B 0,C 180,E1 -28661.565,E2 -28661.565} C_VEL
LIN {X 0,Y 68.671,Z 764.722,A -85,B 0,C 180,E1 -28668.302,E2 -28668.302} C_VEL
LIN {X 0,Y 63.114,Z 767.567,A -85,B 0,C 180,E1 -28676.168,E2 -28676.168} C_VEL
LIN {X 0,Y 60.25,Z 768.9,A -85,B 0,C 180,E1 -28682.188,E2 -28682.188} C_VEL
LIN {X 0,Y 56.454,Z 770.399,A -85,B 0,C 180,E1 -28695.583,E2 -28695.583} C_VEL
LIN {X 0,Y 55.615,Z 770.537,A -85,B 0,C 180,E1 -28702.74,E2 -28702.74} C_VEL
LIN {X 0,Y 55.521,Z 770.268,A -85,B 0,C 180,E1 -28710,E2 -28710} C_VEL
LIN {X 0,Y 56.094,Z 769.622,A -85,B 0,C 180,E1 -28717.197,E2 -28717.197} C_VEL
LIN {X 0,Y 57.268,Z 768.595,A -85,B 0,C 180,E1 -28724.208,E2 -28724.208} C_VEL
LIN {X 0,Y 59.086,Z 767.122,A -85,B 0,C 180,E1 -28730.906,E2 -28730.906} C_VEL
LIN {X 0,Y 63.107,Z 764.129,A -85,B 0,C 180,E1 -28740.075,E2 -28740.075} C_VEL
LIN {X 0,Y 68.461,Z 760.083,A -85,B 0,C 180,E1 -28748.019,E2 -28748.019} C_VEL
LIN {X 0,Y 76.035,Z 753.877,A -85,B 0,C 180,E1 -28755.751,E2 -28755.751} C_VEL
LIN {X 0,Y 82.083,Z 748.314,A -85,B 0,C 180,E1 -28760.405,E2 -28760.405} C_VEL
LIN {X 0,Y 80.658,Z 747.975,A -85,B 0,C 180,E1 -28762.413,E2 -28762.413} C_VEL
LIN {X 0,Y 72.997,Z 748.468,A -85,B 0,C 180,E1 -28771.222,E2 -28771.222} C_VEL
LIN {X 0,Y 70.65,Z 748.162,A -85,B 0,C 180,E1 -28776.551,E2 -28776.551} C_VEL
LIN {X 0,Y 67.901,Z 748.619,A -85,B 0,C 180,E1 -28781.908,E2 -28781.908} C_VEL
LIN {X 0,Y 66.931,Z 748.269,A -85,B 0,C 180,E1 -28787.876,E2 -28787.876} C_VEL
LIN {X 0,Y 65.938,Z 748.452,A -85,B 0,C 180,E1 -28793.88,E2 -28793.88} C_VEL
LIN {X 0,Y 66.452,Z 748.077,A -85,B 0,C 180,E1 -28799.999,E2 -28799.999} C_VEL
LIN {X 0,Y 67.158,Z 748.097,A -85,B 0,C 180,E1 -28806.006,E2 -28806.006} C_VEL
LIN {X 0,Y 69.216,Z 747.625,A -85,B 0,C 180,E1 -28811.715,E2 -28811.715} C_VEL
LIN {X 0,Y 71.496,Z 747.488,A -85,B 0,C 180,E1 -28817.15,E2 -28817.15} C_VEL
LIN {X 0,Y 74.981,Z 746.856,A -85,B 0,C 180,E1 -28822.018,E2 -28822.018} C_VEL
LIN {X 0,Y 79.21,Z 746.603,A -85,B 0,C 180,E1 -28827.472,E2 -28827.472} C_VEL
LIN {X 0,Y 83.016,Z 745.861,A -85,B 0,C 180,E1 -28830.526,E2 -28830.526} C_VEL
LIN {X 0,Y 86.386,Z 745.679,A -85,B 0,C 180,E1 -28833.546,E2 -28833.546} C_VEL
LIN {X 0,Y 85.543,Z 747.082,A -85,B 0,C 180,E1 -28834.76,E2 -28834.76} C_VEL
LIN {X 0,Y 78.371,Z 753.709,A -85,B 0,C 180,E1 -28838.953,E2 -28838.953} C_VEL
LIN {X 0,Y 70.479,Z 760.413,A -85,B 0,C 180,E1 -28845.733,E2 -28845.733} C_VEL
LIN {X 0,Y 64.557,Z 765.101,A -85,B 0,C 180,E1 -28853.22,E2 -28853.22} C_VEL
LIN {X 0,Y 59.875,Z 768.667,A -85,B 0,C 180,E1 -28861.998,E2 -28861.998} C_VEL
LIN {X 0,Y 57.717,Z 770.49,A -85,B 0,C 180,E1 -28868.575,E2 -28868.575} C_VEL
LIN {X 0,Y 56.266,Z 771.85,A -85,B 0,C 180,E1 -28875.534,E2 -28875.534} C_VEL
LIN {X 0,Y 55.537,Z 772.813,A -85,B 0,C 180,E1 -28882.73,E2 -28882.73} C_VEL
LIN {X 0,Y 55.51,Z 773.383,A -85,B 0,C 180,E1 -28890,E2 -28890} C_VEL
LIN {X 0,Y 55.562,Z 773.501,A -85,B 0,C 180,E1 -28897.267,E2 -28897.267} C_VEL
LIN {X 0,Y 57.775,Z 772.534,A -85,B 0,C 180,E1 -28911.403,E2 -28911.403} C_VEL
LIN {X 0,Y 59.98,Z 771.465,A -85,B 0,C 180,E1 -28917.948,E2 -28917.948} C_VEL
LIN {X 0,Y 62.908,Z 769.943,A -85,B 0,C 180,E1 -28923.958,E2 -28923.958} C_VEL
LIN {X 0,Y 68.536,Z 766.88,A -85,B 0,C 180,E1 -28931.799,E2 -28931.799} C_VEL
LIN {X 0,Y 75.209,Z 762.759,A -85,B 0,C 180,E1 -28938.379,E2 -28938.379} C_VEL
LIN {X 0,Y 83.914,Z 756.453,A -85,B 0,C 180,E1 -28944.742,E2 -28944.742} C_VEL
LIN {X 0,Y 92.108,Z 749.581,A -85,B 0,C 180,E1 -28949.135,E2 -28949.135} C_VEL
LIN {X 0,Y 100.809,Z 740.964,A -85,B 0,C 180,E1 -28952.73,E2 -28952.73} C_VEL
LIN {X 0,Y 108.324,Z 732.136,A -85,B 0,C 180,E1 -28955.27,E2 -28955.27} C_VEL
LIN {X 0,Y 115.277,Z 722.436,A -85,B 0,C 180,E1 -28957.233,E2 -28957.233} C_VEL
LIN {X 0,Y 121.571,Z 711.71,A -85,B 0,C 180,E1 -28958.774,E2 -28958.774} C_VEL
LIN {X 0,Y 127.147,Z 699.738,A -85,B 0,C 180,E1 -28959.992,E2 -28959.992} C_VEL
LIN {X 0,Y 131.48,Z 687.49,A -85,B 0,C 180,E1 -28960.875,E2 -28960.875} C_VEL
LIN {X 0,Y 134.618,Z 674.612,A -85,B 0,C 180,E1 -28961.489,E2 -28961.489} C_VEL
LIN {X 0,Y 135.279,Z 671.047,A -85,B 0,C 180,E1 -28961.618,E2 -28961.618} C_VEL
LIN {X 0,Y 135.676,Z 667.205,A -85,B 0,C 180,E1 -28962.049,E2 -28962.049} C_VEL
LIN {X 0,Y 135.45,Z 655.258,A -85,B 0,C 180,E1 -28964.716,E2 -28964.716} C_VEL
LIN {X 0,Y 135.704,Z 651.378,A -85,B 0,C 180,E1 -28965.07,E2 -28965.07} C_VEL
LIN {X 0,Y 135.944,Z 648.777,A -85,B 0,C 180,E1 -28965.221,E2 -28965.221} C_VEL
LIN {X 0,Y 134.667,Z 644.726,A -85,B 0,C 180,E1 -28968.74,E2 -28968.74} C_VEL
LIN {X 0,Y 133.971,Z 642.555,A -85,B 0,C 180,E1 -28971.326,E2 -28971.326} C_VEL
LIN {X 0,Y 133.36,Z 640.164,A -85,B 0,C 180,E1 -28975.088,E2 -28975.088} C_VEL
LIN {X 0,Y 133.134,Z 639.44,A -85,B 0,C 180,E1 -28978.328,E2 -28978.328} C_VEL
LIN {X 0,Y 133.159,Z 639.588,A -85,B 0,C 180,E1 -28980.757,E2 -28980.757} C_VEL
LIN {X 0,Y 133.433,Z 640.529,A -85,B 0,C 180,E1 -28983.776,E2 -28983.776} C_VEL
LIN {X 0,Y 134.178,Z 643.181,A -85,B 0,C 180,E1 -28987.714,E2 -28987.714} C_VEL
LIN {X 0,Y 135.411,Z 647.378,A -85,B 0,C 180,E1 -28991.698,E2 -28991.698} C_VEL
LIN {X 0,Y 135.983,Z 649.531,A -85,B 0,C 180,E1 -28993.198,E2 -28993.198} C_VEL
LIN {X 0,Y 133.475,Z 669.926,A -85,B 0,C 180,E1 -28993.809,E2 -28993.809} C_VEL
LIN {X 0,Y 130.308,Z 683.596,A -85,B 0,C 180,E1 -28994.422,E2 -28994.422} C_VEL
LIN {X 0,Y 126.116,Z 695.957,A -85,B 0,C 180,E1 -28995.26,E2 -28995.26} C_VEL
LIN {X 0,Y 120.884,Z 707.488,A -85,B 0,C 180,E1 -28996.411,E2 -28996.411} C_VEL
LIN {X 0,Y 114.838,Z 718.085,A -85,B 0,C 180,E1 -28997.871,E2 -28997.871} C_VEL
LIN {X 0,Y 107.45,Z 728.656,A -85,B 0,C 180,E1 -28999.914,E2 -28999.914} C_VEL
LIN {X 0,Y 98.882,Z 738.468,A -85,B 0,C 180,E1 -29002.49,E2 -29002.49} C_VEL
LIN {X 0,Y 89.878,Z 747.086,A -85,B 0,C 180,E1 -29005.945,E2 -29005.945} C_VEL
LIN {X 0,Y 81.21,Z 753.947,A -85,B 0,C 180,E1 -29010.072,E2 -29010.072} C_VEL
LIN {X 0,Y 73.103,Z 759.424,A -85,B 0,C 180,E1 -29015.23,E2 -29015.23} C_VEL
LIN {X 0,Y 65.778,Z 763.677,A -85,B 0,C 180,E1 -29021.592,E2 -29021.592} C_VEL
LIN {X 0,Y 61.341,Z 765.921,A -85,B 0,C 180,E1 -29026.574,E2 -29026.574} C_VEL
LIN {X 0,Y 57.328,Z 767.732,A -85,B 0,C 180,E1 -29032.197,E2 -29032.197} C_VEL
LIN {X 0,Y 51.433,Z 770.019,A -85,B 0,C 180,E1 -29045.8,E2 -29045.8} C_VEL
LIN {X 0,Y 49.589,Z 770.582,A -85,B 0,C 180,E1 -29053.534,E2 -29053.534} C_VEL
LIN {X 0,Y 48.585,Z 770.731,A -85,B 0,C 180,E1 -29061.683,E2 -29061.683} C_VEL
LIN {X 0,Y 48.439,Z 770.467,A -85,B 0,C 180,E1 -29070,E2 -29070} C_VEL
LIN {X 0,Y 49.074,Z 769.826,A -85,B 0,C 180,E1 -29078.234,E2 -29078.234} C_VEL
LIN {X 0,Y 50.435,Z 768.806,A -85,B 0,C 180,E1 -29086.182,E2 -29086.182} C_VEL
LIN {X 0,Y 52.52,Z 767.343,A -85,B 0,C 180,E1 -29093.668,E2 -29093.668} C_VEL
LIN {X 0,Y 57.075,Z 764.362,A -85,B 0,C 180,E1 -29103.649,E2 -29103.649} C_VEL
LIN {X 0,Y 63.025,Z 760.328,A -85,B 0,C 180,E1 -29111.994,E2 -29111.994} C_VEL
LIN {X 0,Y 70.013,Z 755.125,A -85,B 0,C 180,E1 -29118.837,E2 -29118.837} C_VEL
LIN {X 0,Y 73.464,Z 752.355,A -85,B 0,C 180,E1 -29121.463,E2 -29121.463} C_VEL
LIN {X 0,Y 72.851,Z 752.047,A -85,B 0,C 180,E1 -29122.844,E2 -29122.844} C_VEL
LIN {X 0,Y 67.879,Z 752.37,A -85,B 0,C 180,E1 -29128.821,E2 -29128.821} C_VEL
LIN {X 0,Y 65.256,Z 752.121,A -85,B 0,C 180,E1 -29134.48,E2 -29134.48} C_VEL
LIN {X 0,Y 62.307,Z 752.546,A -85,B 0,C 180,E1 -29140.22,E2 -29140.22} C_VEL
LIN {X 0,Y 61.137,Z 752.264,A -85,B 0,C 180,E1 -29146.707,E2 -29146.707} C_VEL
LIN {X 0,Y 60.106,Z 752.403,A -85,B 0,C 180,E1 -29153.284,E2 -29153.284} C_VEL
LIN {X 0,Y 60.556,Z 752.124,A -85,B 0,C 180,E1 -29159.998,E2 -29159.998} C_VEL
LIN {X 0,Y 61.365,Z 752.131,A -85,B 0,C 180,E1 -29166.575,E2 -29166.575} C_VEL
LIN {X 0,Y 63.507,Z 751.766,A -85,B 0,C 180,E1 -29172.786,E2 -29172.786} C_VEL
LIN {X 0,Y 65.984,Z 751.627,A -85,B 0,C 180,E1 -29178.633,E2 -29178.633} C_VEL
LIN {X 0,Y 69.618,Z 751.089,A -85,B 0,C 180,E1 -29183.815,E2 -29183.815} C_VEL
LIN {X 0,Y 75.544,Z 750.667,A -85,B 0,C 180,E1 -29190.809,E2 -29190.809} C_VEL
LIN {X 0,Y 76.714,Z 750.474,A -85,B 0,C 180,E1 -29191.723,E2 -29191.723} C_VEL
LIN {X 0,Y 75.915,Z 751.922,A -85,B 0,C 180,E1 -29193.574,E2 -29193.574} C_VEL
LIN {X 0,Y 69.261,Z 757.353,A -85,B 0,C 180,E1 -29198.152,E2 -29198.152} C_VEL
LIN {X 0,Y 61.068,Z 763.441,A -85,B 0,C 180,E1 -29206.331,E2 -29206.331} C_VEL
LIN {X 0,Y 55.294,Z 767.376,A -85,B 0,C 180,E1 -29215.114,E2 -29215.114} C_VEL
LIN {X 0,Y 51.129,Z 770.272,A -85,B 0,C 180,E1 -29225.647,E2 -29225.647} C_VEL
LIN {X 0,Y 49.385,Z 771.64,A -85,B 0,C 180,E1 -29233.464,E2 -29233.464} C_VEL
LIN {X 0,Y 48.491,Z 772.609,A -85,B 0,C 180,E1 -29241.667,E2 -29241.667} C_VEL
LIN {X 0,Y 48.427,Z 773.185,A -85,B 0,C 180,E1 -29250,E2 -29250} C_VEL
LIN {X 0,Y 48.511,Z 773.312,A -85,B 0,C 180,E1 -29258.33,E2 -29258.33} C_VEL
LIN {X 0,Y 51.189,Z 772.356,A -85,B 0,C 180,E1 -29274.323,E2 -29274.323} C_VEL
LIN {X 0,Y 53.773,Z 771.294,A -85,B 0,C 180,E1 -29281.519,E2 -29281.519} C_VEL
LIN {X 0,Y 57.144,Z 769.782,A -85,B 0,C 180,E1 -29287.946,E2 -29287.946} C_VEL
LIN {X 0,Y 63.387,Z 766.731,A -85,B 0,C 180,E1 -29296.11,E2 -29296.11} C_VEL
LIN {X 0,Y 70.666,Z 762.623,A -85,B 0,C 180,E1 -29302.713,E2 -29302.713} C_VEL
LIN {X 0,Y 80.001,Z 756.331,A -85,B 0,C 180,E1 -29308.926,E2 -29308.926} C_VEL
LIN {X 0,Y 88.673,Z 749.48,A -85,B 0,C 180,E1 -29313.079,E2 -29313.079} C_VEL
LIN {X 0,Y 97.76,Z 740.887,A -85,B 0,C 180,E1 -29316.431,E2 -29316.431} C_VEL
LIN {X 0,Y 105.548,Z 732.083,A -85,B 0,C 180,E1 -29318.777,E2 -29318.777} C_VEL
LIN {X 0,Y 112.725,Z 722.412,A -85,B 0,C 180,E1 -29320.556,E2 -29320.556} C_VEL
LIN {X 0,Y 119.191,Z 711.745,A -85,B 0,C 180,E1 -29321.948,E2 -29321.948} C_VEL
LIN {X 0,Y 124.901,Z 699.833,A -85,B 0,C 180,E1 -29323.046,E2 -29323.046} C_VEL
LIN {X 0,Y 129.068,Z 688.463,A -85,B 0,C 180,E1 -29323.812,E2 -29323.812} C_VEL
LIN {X 0,Y 132.312,Z 676.232,A -85,B 0,C 180,E1 -29324.358,E2 -29324.358} C_VEL
LIN {X 0,Y 134.476,Z 662.352,A -85,B 0,C 180,E1 -29324.8,E2 -29324.8} C_VEL
LIN {X 0,Y 135.704,Z 651.378,A -85,B 0,C 180,E1 -29325.07,E2 -29325.07} C_VEL
LIN {X 0,Y 135.71,Z 649.748,A -85,B 0,C 180,E1 -29325.413,E2 -29325.413} C_VEL
LIN {X 0,Y 135.375,Z 648.449,A -85,B 0,C 180,E1 -29326.309,E2 -29326.309} C_VEL
LIN {X 0,Y 134.662,Z 647.815,A -85,B 0,C 180,E1 -29327.89,E2 -29327.89} C_VEL
LIN {X 0,Y 132.848,Z 648.636,A -85,B 0,C 180,E1 -29332.594,E2 -29332.594} C_VEL
LIN {X 0,Y 132.585,Z 648.133,A -85,B 0,C 180,E1 -29333.972,E2 -29333.972} C_VEL
LIN {X 0,Y 132.443,Z 647.173,A -85,B 0,C 180,E1 -29335.435,E2 -29335.435} C_VEL
LIN {X 0,Y 132.264,Z 646.484,A -85,B 0,C 180,E1 -29338.478,E2 -29338.478} C_VEL
LIN {X 0,Y 132.289,Z 646.673,A -85,B 0,C 180,E1 -29340.762,E2 -29340.762} C_VEL
LIN {X 0,Y 132.479,Z 647.48,A -85,B 0,C 180,E1 -29343.232,E2 -29343.232} C_VEL
LIN {X 0,Y 133.046,Z 649.906,A -85,B 0,C 180,E1 -29346.827,E2 -29346.827} C_VEL
LIN {X 0,Y 133.966,Z 653.562,A -85,B 0,C 180,E1 -29350.355,E2 -29350.355} C_VEL
LIN {X 0,Y 131.693,Z 670.787,A -85,B 0,C 180,E1 -29350.842,E2 -29350.842} C_VEL
LIN {X 0,Y 128.408,Z 684.44,A -85,B 0,C 180,E1 -29351.41,E2 -29351.41} C_VEL
LIN {X 0,Y 123.947,Z 696.993,A -85,B 0,C 180,E1 -29352.184,E2 -29352.184} C_VEL
LIN {X 0,Y 118.246,Z 708.991,A -85,B 0,C 180,E1 -29353.287,E2 -29353.287} C_VEL
LIN {X 0,Y 112.522,Z 718.612,A -85,B 0,C 180,E1 -29354.509,E2 -29354.509} C_VEL
LIN {X 0,Y 105.245,Z 728.699,A -85,B 0,C 180,E1 -29356.281,E2 -29356.281} C_VEL
LIN {X 0,Y 96.387,Z 738.543,A -85,B 0,C 180,E1 -29358.582,E2 -29358.582} C_VEL
LIN {X 0,Y 86.996,Z 747.182,A -85,B 0,C 180,E1 -29361.719,E2 -29361.719} C_VEL
LIN {X 0,Y 77.88,Z 754.067,A -85,B 0,C 180,E1 -29365.526,E2 -29365.526} C_VEL
LIN {X 0,Y 68.551,Z 759.945,A -85,B 0,C 180,E1 -29370.84,E2 -29370.84} C_VEL
LIN {X 0,Y 58.793,Z 765.029,A -85,B 0,C 180,E1 -29379.015,E2 -29379.015} C_VEL
LIN {X 0,Y 51.88,Z 767.896,A -85,B 0,C 180,E1 -29387.366,E2 -29387.366} C_VEL
LIN {X 0,Y 48.1,Z 769.244,A -85,B 0,C 180,E1 -29394.237,E2 -29394.237} C_VEL
LIN {X 0,Y 42.818,Z 770.765,A -85,B 0,C 180,E1 -29410.836,E2 -29410.836} C_VEL
LIN {X 0,Y 41.566,Z 770.925,A -85,B 0,C 180,E1 -29420.266,E2 -29420.266} C_VEL
LIN {X 0,Y 41.34,Z 770.666,A -85,B 0,C 180,E1 -29430,E2 -29430} C_VEL
LIN {X 0,Y 42.064,Z 770.031,A -85,B 0,C 180,E1 -29439.618,E2 -29439.618} C_VEL
LIN {X 0,Y 43.664,Z 769.016,A -85,B 0,C 180,E1 -29448.778,E2 -29448.778} C_VEL
LIN {X 0,Y 46.121,Z 767.564,A -85,B 0,C 180,E1 -29457.203,E2 -29457.203} C_VEL
LIN {X 0,Y 51.323,Z 764.595,A -85,B 0,C 180,E1 -29468.039,E2 -29468.039} C_VEL
LIN {X 0,Y 57.953,Z 760.573,A -85,B 0,C 180,E1 -29476.686,E2 -29476.686} C_VEL
LIN {X 0,Y 64.082,Z 756.459,A -85,B 0,C 180,E1 -29482.367,E2 -29482.367} C_VEL
LIN {X 0,Y 63.888,Z 755.88,A -85,B 0,C 180,E1 -29484.397,E2 -29484.397} C_VEL
LIN {X 0,Y 59.775,Z 755.754,A -85,B 0,C 180,E1 -29491.945,E2 -29491.945} C_VEL
LIN {X 0,Y 56.606,Z 756.133,A -85,B 0,C 180,E1 -29498.13,E2 -29498.13} C_VEL
LIN {X 0,Y 55.194,Z 755.912,A -85,B 0,C 180,E1 -29505.245,E2 -29505.245} C_VEL
LIN {X 0,Y 54.077,Z 756.029,A -85,B 0,C 180,E1 -29512.531,E2 -29512.531} C_VEL
LIN {X 0,Y 54.442,Z 755.818,A -85,B 0,C 180,E1 -29519.998,E2 -29519.998} C_VEL
LIN {X 0,Y 55.334,Z 755.821,A -85,B 0,C 180,E1 -29527.295,E2 -29527.295} C_VEL
LIN {X 0,Y 60.301,Z 755.418,A -85,B 0,C 180,E1 -29540.464,E2 -29540.464} C_VEL
LIN {X 0,Y 64.12,Z 755.004,A -85,B 0,C 180,E1 -29546.002,E2 -29546.002} C_VEL
LIN {X 0,Y 68.16,Z 754.779,A -85,B 0,C 180,E1 -29551.033,E2 -29551.033} C_VEL
LIN {X 0,Y 61.105,Z 759.912,A -85,B 0,C 180,E1 -29556.381,E2 -29556.381} C_VEL
LIN {X 0,Y 53.812,Z 764.623,A -85,B 0,C 180,E1 -29564.086,E2 -29564.086} C_VEL
LIN {X 0,Y 47.74,Z 768.212,A -85,B 0,C 180,E1 -29573.925,E2 -29573.925} C_VEL
LIN {X 0,Y 44.722,Z 770.055,A -85,B 0,C 180,E1 -29581.873,E2 -29581.873} C_VEL
LIN {X 0,Y 42.6,Z 771.429,A -85,B 0,C 180,E1 -29590.734,E2 -29590.734} C_VEL
LIN {X 0,Y 41.46,Z 772.404,A -85,B 0,C 180,E1 -29600.241,E2 -29600.241} C_VEL
LIN {X 0,Y 41.326,Z 772.986,A -85,B 0,C 180,E1 -29610,E2 -29610} C_VEL
LIN {X 0,Y 41.477,Z 773.123,A -85,B 0,C 180,E1 -29619.755,E2 -29619.755} C_VEL
LIN {X 0,Y 44.781,Z 772.177,A -85,B 0,C 180,E1 -29638.087,E2 -29638.087} C_VEL
LIN {X 0,Y 47.83,Z 771.123,A -85,B 0,C 180,E1 -29645.996,E2 -29645.996} C_VEL
LIN {X 0,Y 51.722,Z 769.622,A -85,B 0,C 180,E1 -29652.796,E2 -29652.796} C_VEL
LIN {X 0,Y 58.661,Z 766.581,A -85,B 0,C 180,E1 -29661.144,E2 -29661.144} C_VEL
LIN {X 0,Y 66.582,Z 762.487,A -85,B 0,C 180,E1 -29667.609,E2 -29667.609} C_VEL
LIN {X 0,Y 76.564,Z 756.21,A -85,B 0,C 180,E1 -29673.503,E2 -29673.503} C_VEL
LIN {X 0,Y 85.691,Z 749.377,A -85,B 0,C 180,E1 -29677.318,E2 -29677.318} C_VEL
LIN {X 0,Y 95.146,Z 740.811,A -85,B 0,C 180,E1 -29680.349,E2 -29680.349} C_VEL
LIN {X 0,Y 103.19,Z 732.03,A -85,B 0,C 180,E1 -29682.455,E2 -29682.455} C_VEL
LIN {X 0,Y 110.566,Z 722.389,A -85,B 0,C 180,E1 -29684.024,E2 -29684.024} C_VEL
LIN {X 0,Y 117.19,Z 711.78,A -85,B 0,C 180,E1 -29685.241,E2 -29685.241} C_VEL
LIN {X 0,Y 123.023,Z 699.927,A -85,B 0,C 180,E1 -29686.203,E2 -29686.203} C_VEL
LIN {X 0,Y 127.452,Z 688.116,A -85,B 0,C 180,E1 -29686.902,E2 -29686.902} C_VEL
LIN {X 0,Y 130.793,Z 675.611,A -85,B 0,C 180,E1 -29687.381,E2 -29687.381} C_VEL
LIN {X 0,Y 133.102,Z 660.584,A -85,B 0,C 180,E1 -29687.808,E2 -29687.808} C_VEL
LIN {X 0,Y 133.936,Z 653.131,A -85,B 0,C 180,E1 -29688.021,E2 -29688.021} C_VEL
LIN {X 0,Y 132.954,Z 649.504,A -85,B 0,C 180,E1 -29691.833,E2 -29691.833} C_VEL
LIN {X 0,Y 132.585,Z 648.133,A -85,B 0,C 180,E1 -29693.972,E2 -29693.972} C_VEL
LIN {X 0,Y 132.326,Z 647.882,A -85,B 0,C 180,E1 -29695.64,E2 -29695.64} C_VEL
LIN {X 0,Y 132.033,Z 648.833,A -85,B 0,C 180,E1 -29697.299,E2 -29697.299} C_VEL
LIN {X 0,Y 131.518,Z 654.075,A -85,B 0,C 180,E1 -29702.209,E2 -29702.209} C_VEL
LIN {X 0,Y 131.546,Z 654.495,A -85,B 0,C 180,E1 -29702.788,E2 -29702.788} C_VEL
LIN {X 0,Y 131.95,Z 656.605,A -85,B 0,C 180,E1 -29705.924,E2 -29705.924} C_VEL
LIN {X 0,Y 132.241,Z 658.103,A -85,B 0,C 180,E1 -29707.474,E2 -29707.474} C_VEL
LIN {X 0,Y 129.947,Z 673.323,A -85,B 0,C 180,E1 -29707.875,E2 -29707.875} C_VEL
LIN {X 0,Y 126.601,Z 686.168,A -85,B 0,C 180,E1 -29708.358,E2 -29708.358} C_VEL
LIN {X 0,Y 121.754,Z 698.923,A -85,B 0,C 180,E1 -29709.07,E2 -29709.07} C_VEL
LIN {X 0,Y 115.974,Z 710.496,A -85,B 0,C 180,E1 -29710.028,E2 -29710.028} C_VEL
LIN {X 0,Y 109.268,Z 721.116,A -85,B 0,C 180,E1 -29711.319,E2 -29711.319} C_VEL
LIN {X 0,Y 100.98,Z 731.639,A -85,B 0,C 180,E1 -29713.007,E2 -29713.007} C_VEL
LIN {X 0,Y 92.723,Z 740.216,A -85,B 0,C 180,E1 -29714.901,E2 -29714.901} C_VEL
LIN {X 0,Y 83.017,Z 748.523,A -85,B 0,C 180,E1 -29717.755,E2 -29717.755} C_VEL
LIN {X 0,Y 75.089,Z 754.187,A -85,B 0,C 180,E1 -29720.62,E2 -29720.62} C_VEL
LIN {X 0,Y 64.456,Z 760.467,A -85,B 0,C 180,E1 -29725.86,E2 -29725.86} C_VEL
LIN {X 0,Y 54.586,Z 765.181,A -85,B 0,C 180,E1 -29733.189,E2 -29733.189} C_VEL
LIN {X 0,Y 46.889,Z 768.059,A -85,B 0,C 180,E1 -29741.46,E2 -29741.46} C_VEL
LIN {X 0,Y 38.887,Z 770.374,A -85,B 0,C 180,E1 -29757.168,E2 -29757.168} C_VEL
LIN {X 0,Y 36.186,Z 770.948,A -85,B 0,C 180,E1 -29767.143,E2 -29767.143} C_VEL
LIN {X 0,Y 34.576,Z 771.119,A -85,B 0,C 180,E1 -29778.273,E2 -29778.273} C_VEL
LIN {X 0,Y 34.256,Z 770.865,A -85,B 0,C 180,E1 -29790,E2 -29790} C_VEL
LIN {X 0,Y 35.106,Z 770.235,A -85,B 0,C 180,E1 -29801.548,E2 -29801.548} C_VEL
LIN {X 0,Y 37.029,Z 769.226,A -85,B 0,C 180,E1 -29812.308,E2 -29812.308} C_VEL
LIN {X 0,Y 39.942,Z 767.785,A -85,B 0,C 180,E1 -29821.861,E2 -29821.861} C_VEL
LIN {X 0,Y 45.952,Z 764.827,A -85,B 0,C 180,E1 -29833.489,E2 -29833.489} C_VEL
LIN {X 0,Y 53.346,Z 760.817,A -85,B 0,C 180,E1 -29842.228,E2 -29842.228} C_VEL
LIN {X 0,Y 55.591,Z 759.485,A -85,B 0,C 180,E1 -29844.262,E2 -29844.262} C_VEL
LIN {X 0,Y 55.272,Z 759.083,A -85,B 0,C 180,E1 -29846.639,E2 -29846.639} C_VEL
LIN {X 0,Y 54.267,Z 759.043,A -85,B 0,C 180,E1 -29848.797,E2 -29848.797} C_VEL
LIN {X 0,Y 50.811,Z 759.376,A -85,B 0,C 180,E1 -29855.482,E2 -29855.482} C_VEL
LIN {X 0,Y 49.111,Z 759.223,A -85,B 0,C 180,E1 -29863.367,E2 -29863.367} C_VEL
LIN {X 0,Y 47.852,Z 759.331,A -85,B 0,C 180,E1 -29871.552,E2 -29871.552} C_VEL
LIN {X 0,Y 50.524,Z 759.04,A -85,B 0,C 180,E1 -29893.171,E2 -29893.171} C_VEL
LIN {X 0,Y 58.541,Z 758.528,A -85,B 0,C 180,E1 -29908.697,E2 -29908.697} C_VEL
LIN {X 0,Y 57.173,Z 759.661,A -85,B 0,C 180,E1 -29910.632,E2 -29910.632} C_VEL
LIN {X 0,Y 49.117,Z 764.384,A -85,B 0,C 180,E1 -29918.098,E2 -29918.098} C_VEL
LIN {X 0,Y 42.18,Z 767.984,A -85,B 0,C 180,E1 -29928.206,E2 -29928.206} C_VEL
LIN {X 0,Y 38.582,Z 769.837,A -85,B 0,C 180,E1 -29936.875,E2 -29936.875} C_VEL
LIN {X 0,Y 35.956,Z 771.219,A -85,B 0,C 180,E1 -29946.989,E2 -29946.989} C_VEL
LIN {X 0,Y 34.478,Z 772.199,A -85,B 0,C 180,E1 -29958.239,E2 -29958.239} C_VEL
LIN {X 0,Y 34.24,Z 772.787,A -85,B 0,C 180,E1 -29970,E2 -29970} C_VEL
LIN {X 0,Y 34.492,Z 772.935,A -85,B 0,C 180,E1 -29981.756,E2 -29981.756} C_VEL
LIN {X 0,Y 38.637,Z 771.999,A -85,B 0,C 180,E1 -30003.071,E2 -30003.071} C_VEL
LIN {X 0,Y 42.263,Z 770.951,A -85,B 0,C 180,E1 -30011.694,E2 -30011.694} C_VEL
LIN {X 0,Y 46.756,Z 769.461,A -85,B 0,C 180,E1 -30018.725,E2 -30018.725} C_VEL
LIN {X 0,Y 54.47,Z 766.432,A -85,B 0,C 180,E1 -30026.997,E2 -30026.997} C_VEL
LIN {X 0,Y 63.04,Z 762.35,A -85,B 0,C 180,E1 -30033.107,E2 -30033.107} C_VEL
LIN {X 0,Y 73.662,Z 756.089,A -85,B 0,C 180,E1 -30038.468,E2 -30038.468} C_VEL
LIN {X 0,Y 83.203,Z 749.273,A -85,B 0,C 180,E1 -30041.85,E2 -30041.85} C_VEL
LIN {X 0,Y 93,Z 740.735,A -85,B 0,C 180,E1 -30044.471,E2 -30044.471} C_VEL
LIN {X 0,Y 101.277,Z 731.978,A -85,B 0,C 180,E1 -30046.286,E2 -30046.286} C_VEL
LIN {X 0,Y 108.828,Z 722.365,A -85,B 0,C 180,E1 -30047.615,E2 -30047.615} C_VEL
